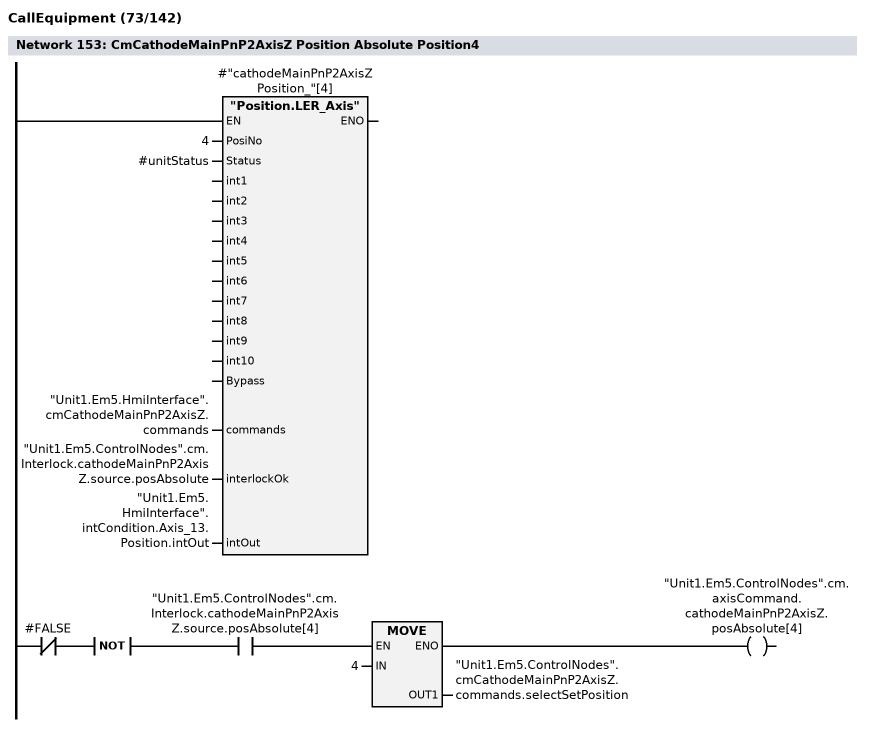
   RUNG wire#powerrail
      #"cathodeMainPnP2AxisZ Position_"[4](PosiNo := 4, Status := #unitStatus, int1 :=, int2 :=, int3 :=, int4 :=, int5 :=, int6 :=, int7 :=, int8 :=, int9 :=, int10 :=, Bypass :=, commands := "Unit1.Em5.HmiInterface".cmCathodeMainPnP2AxisZ.commands, interlockOk := "Unit1.Em5.ControlNodes".cm.Interlock.cathodeMainPnP2AxisZ.source.posAbsolute, intOut := "Unit1.Em5.HmiInterface".intCondition.Axis_13.Position.intOut)
   END_RUNG
   RUNG wire#powerrail
      I_Contact( #FALSE )
      Not()
      Contact( "Unit1.Em5.ControlNodes".cm.Interlock.cathodeMainPnP2AxisZ.source.posAbsolute[4] )
      Move(in := 4, out1 => "Unit1.Em5.ControlNodes".cmCathodeMainPnP2AxisZ.commands.selectSetPosition)
      Coil( "Unit1.Em5.ControlNodes".cm.axisCommand.cathodeMainPnP2AxisZ.posAbsolute[4] )
   END_RUNG
   // the same network as SCL:
   #"cathodeMainPnP2AxisZ Position_"[4](PosiNo := 4,   // "Position.LER_Axis"
                           Status := #unitStatus,
                           commands := "Unit1.Em5.HmiInterface".cmCathodeMainPnP2AxisZ.commands,
                           interlockOk := "Unit1.Em5.ControlNodes".cm.Interlock.cathodeMainPnP2AxisZ.source.posAbsolute,
                           intOut := "Unit1.Em5.HmiInterface".intCondition.Axis_13.Position.intOut);
   #_w1 := NOT (NOT #FALSE) AND "Unit1.Em5.ControlNodes".cm.Interlock.cathodeMainPnP2AxisZ.source.posAbsolute[4];
   IF #_w1 THEN "Unit1.Em5.ControlNodes".cmCathodeMainPnP2AxisZ.commands.selectSetPosition := 4; END_IF;
   "Unit1.Em5.ControlNodes".cm.axisCommand.cathodeMainPnP2AxisZ.posAbsolute[4] := #_w1;
END_REGION

REGION Network 154: CmCathodeMainPnP2AxisZ Position Absolute Position5
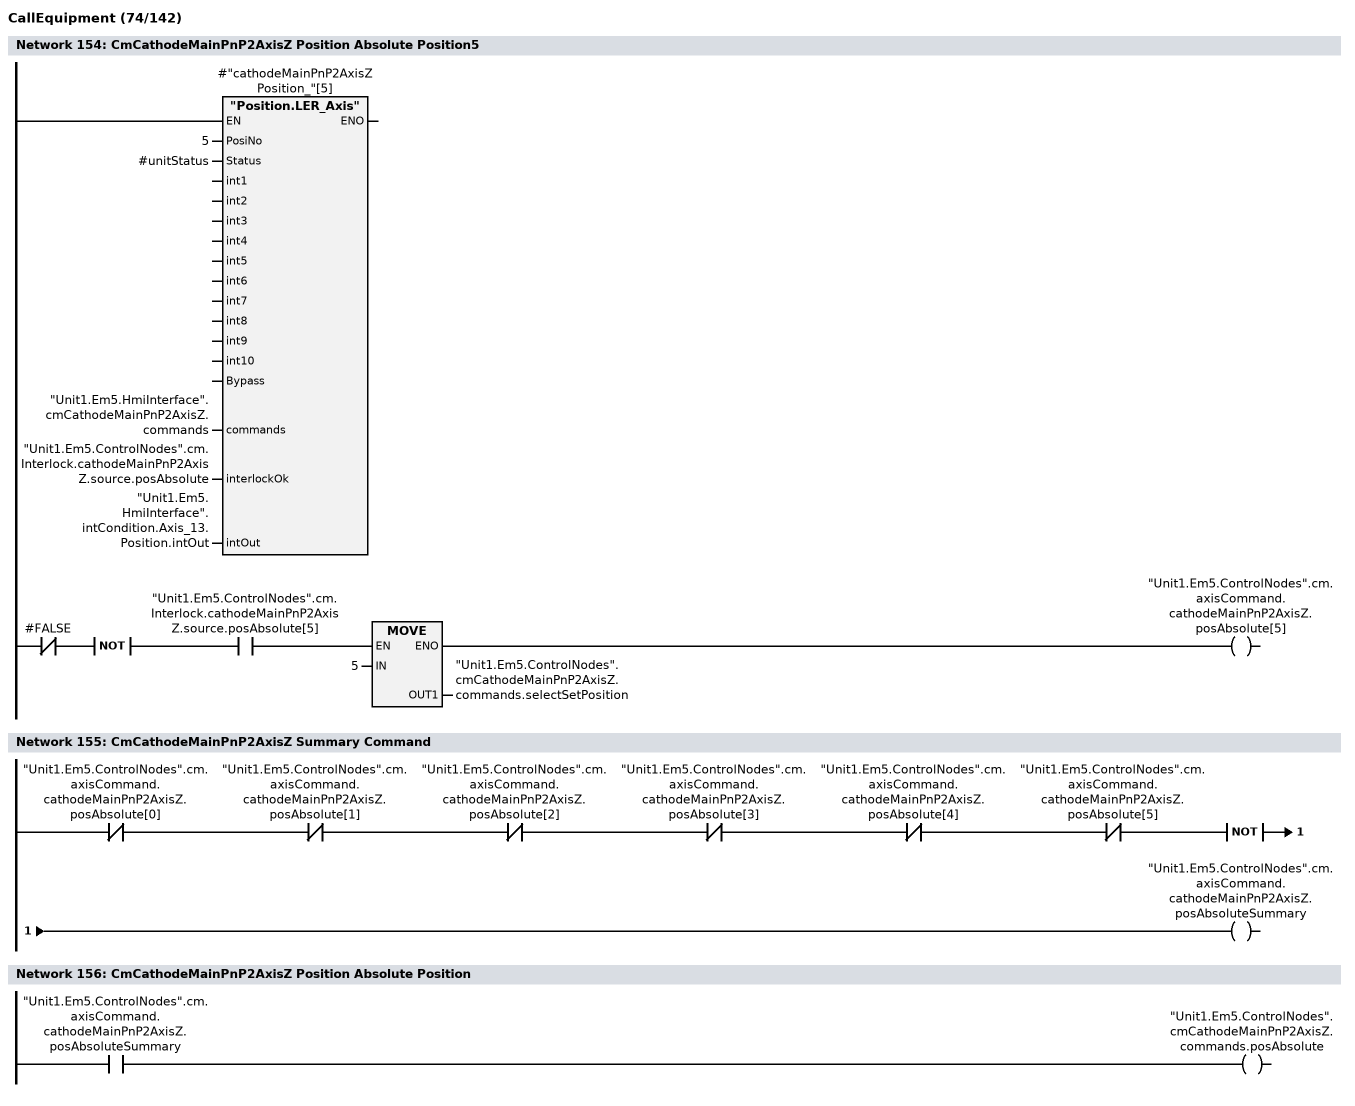
   RUNG wire#powerrail
      #"cathodeMainPnP2AxisZ Position_"[5](PosiNo := 5, Status := #unitStatus, int1 :=, int2 :=, int3 :=, int4 :=, int5 :=, int6 :=, int7 :=, int8 :=, int9 :=, int10 :=, Bypass :=, commands := "Unit1.Em5.HmiInterface".cmCathodeMainPnP2AxisZ.commands, interlockOk := "Unit1.Em5.ControlNodes".cm.Interlock.cathodeMainPnP2AxisZ.source.posAbsolute, intOut := "Unit1.Em5.HmiInterface".intCondition.Axis_13.Position.intOut)
   END_RUNG
   RUNG wire#powerrail
      I_Contact( #FALSE )
      Not()
      Contact( "Unit1.Em5.ControlNodes".cm.Interlock.cathodeMainPnP2AxisZ.source.posAbsolute[5] )
      Move(in := 5, out1 => "Unit1.Em5.ControlNodes".cmCathodeMainPnP2AxisZ.commands.selectSetPosition)
      Coil( "Unit1.Em5.ControlNodes".cm.axisCommand.cathodeMainPnP2AxisZ.posAbsolute[5] )
   END_RUNG
   // the same network as SCL:
   #"cathodeMainPnP2AxisZ Position_"[5](PosiNo := 5,   // "Position.LER_Axis"
                           Status := #unitStatus,
                           commands := "Unit1.Em5.HmiInterface".cmCathodeMainPnP2AxisZ.commands,
                           interlockOk := "Unit1.Em5.ControlNodes".cm.Interlock.cathodeMainPnP2AxisZ.source.posAbsolute,
                           intOut := "Unit1.Em5.HmiInterface".intCondition.Axis_13.Position.intOut);
   #_w1 := NOT (NOT #FALSE) AND "Unit1.Em5.ControlNodes".cm.Interlock.cathodeMainPnP2AxisZ.source.posAbsolute[5];
   IF #_w1 THEN "Unit1.Em5.ControlNodes".cmCathodeMainPnP2AxisZ.commands.selectSetPosition := 5; END_IF;
   "Unit1.Em5.ControlNodes".cm.axisCommand.cathodeMainPnP2AxisZ.posAbsolute[5] := #_w1;
END_REGION

REGION Network 155: CmCathodeMainPnP2AxisZ Summary Command
   RUNG wire#powerrail
      I_Contact( "Unit1.Em5.ControlNodes".cm.axisCommand.cathodeMainPnP2AxisZ.posAbsolute[0] )
      I_Contact( "Unit1.Em5.ControlNodes".cm.axisCommand.cathodeMainPnP2AxisZ.posAbsolute[1] )
      I_Contact( "Unit1.Em5.ControlNodes".cm.axisCommand.cathodeMainPnP2AxisZ.posAbsolute[2] )
      I_Contact( "Unit1.Em5.ControlNodes".cm.axisCommand.cathodeMainPnP2AxisZ.posAbsolute[3] )
      I_Contact( "Unit1.Em5.ControlNodes".cm.axisCommand.cathodeMainPnP2AxisZ.posAbsolute[4] )
      I_Contact( "Unit1.Em5.ControlNodes".cm.axisCommand.cathodeMainPnP2AxisZ.posAbsolute[5] )
      Not()
      Coil( "Unit1.Em5.ControlNodes".cm.axisCommand.cathodeMainPnP2AxisZ.posAbsoluteSummary )
   END_RUNG
   // the same network as SCL:
   "Unit1.Em5.ControlNodes".cm.axisCommand.cathodeMainPnP2AxisZ.posAbsoluteSummary := NOT (NOT "Unit1.Em5.ControlNodes".cm.axisCommand.cathodeMainPnP2AxisZ.posAbsolute[0] AND NOT "Unit1.Em5.ControlNodes".cm.axisCommand.cathodeMainPnP2AxisZ.posAbsolute[1] AND NOT "Unit1.Em5.ControlNodes".cm.axisCommand.cathodeMainPnP2AxisZ.posAbsolute[2] AND NOT "Unit1.Em5.ControlNodes".cm.axisCommand.cathodeMainPnP2AxisZ.posAbsolute[3] AND NOT "Unit1.Em5.ControlNodes".cm.axisCommand.cathodeMainPnP2AxisZ.posAbsolute[4] AND NOT "Unit1.Em5.ControlNodes".cm.axisCommand.cathodeMainPnP2AxisZ.posAbsolute[5]);
END_REGION

REGION Network 156: CmCathodeMainPnP2AxisZ Position Absolute Position
   RUNG wire#powerrail
      Contact( "Unit1.Em5.ControlNodes".cm.axisCommand.cathodeMainPnP2AxisZ.posAbsoluteSummary )
      Coil( "Unit1.Em5.ControlNodes".cmCathodeMainPnP2AxisZ.commands.posAbsolute )
   END_RUNG
   // the same network as SCL:
   "Unit1.Em5.ControlNodes".cmCathodeMainPnP2AxisZ.commands.posAbsolute := "Unit1.Em5.ControlNodes".cm.axisCommand.cathodeMainPnP2AxisZ.posAbsoluteSummary;
END_REGION

REGION Network 157: CmCathodeMainPnP1AxisZ Interlock Summary
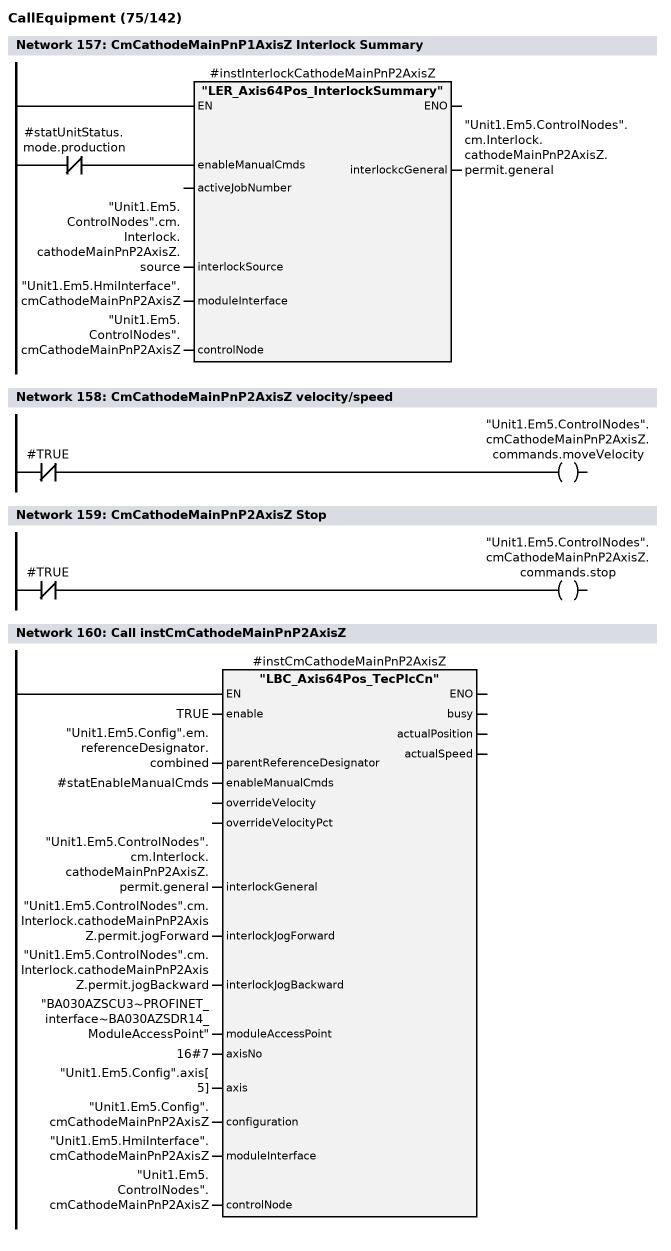
   RUNG wire#powerrail
      #instInterlockCathodeMainPnP2AxisZ(enableManualCmds := wire#w1, activeJobNumber :=, interlockSource := "Unit1.Em5.ControlNodes".cm.Interlock.cathodeMainPnP2AxisZ.source, moduleInterface := "Unit1.Em5.HmiInterface".cmCathodeMainPnP2AxisZ, controlNode := "Unit1.Em5.ControlNodes".cmCathodeMainPnP2AxisZ, interlockcGeneral => "Unit1.Em5.ControlNodes".cm.Interlock.cathodeMainPnP2AxisZ.permit.general)
   END_RUNG
   RUNG wire#powerrail
      I_Contact( #statUnitStatus.mode.production )
   END_RUNG wire#w1
   // the same network as SCL:
   #instInterlockCathodeMainPnP2AxisZ(enableManualCmds := NOT #statUnitStatus.mode.production,   // "LER_Axis64Pos_InterlockSummary"
                           interlockSource := "Unit1.Em5.ControlNodes".cm.Interlock.cathodeMainPnP2AxisZ.source,
                           moduleInterface := "Unit1.Em5.HmiInterface".cmCathodeMainPnP2AxisZ,
                           controlNode := "Unit1.Em5.ControlNodes".cmCathodeMainPnP2AxisZ,
                           interlockcGeneral => "Unit1.Em5.ControlNodes".cm.Interlock.cathodeMainPnP2AxisZ.permit.general);
END_REGION

REGION Network 158: CmCathodeMainPnP2AxisZ velocity/speed
   RUNG wire#powerrail
      I_Contact( #TRUE )
      Coil( "Unit1.Em5.ControlNodes".cmCathodeMainPnP2AxisZ.commands.moveVelocity )
   END_RUNG
   // the same network as SCL:
   "Unit1.Em5.ControlNodes".cmCathodeMainPnP2AxisZ.commands.moveVelocity := NOT #TRUE;
END_REGION

REGION Network 159: CmCathodeMainPnP2AxisZ Stop
   RUNG wire#powerrail
      I_Contact( #TRUE )
      Coil( "Unit1.Em5.ControlNodes".cmCathodeMainPnP2AxisZ.commands.stop )
   END_RUNG
   // the same network as SCL:
   "Unit1.Em5.ControlNodes".cmCathodeMainPnP2AxisZ.commands.stop := NOT #TRUE;
END_REGION

REGION Network 160: Call instCmCathodeMainPnP2AxisZ
   RUNG wire#powerrail
      #instCmCathodeMainPnP2AxisZ(enable := TRUE, parentReferenceDesignator := "Unit1.Em5.Config".em.referenceDesignator.combined, enableManualCmds := #statEnableManualCmds, overrideVelocity :=, overrideVelocityPct :=, interlockGeneral := "Unit1.Em5.ControlNodes".cm.Interlock.cathodeMainPnP2AxisZ.permit.general, interlockJogForward := "Unit1.Em5.ControlNodes".cm.Interlock.cathodeMainPnP2AxisZ.permit.jogForward, interlockJogBackward := "Unit1.Em5.ControlNodes".cm.Interlock.cathodeMainPnP2AxisZ.permit.jogBackward, moduleAccessPoint := "BA030AZSCU3~PROFINET_interface~BA030AZSDR14_ModuleAccessPoint", axisNo := 16#7, axis := "Unit1.Em5.Config".axis[5], configuration := "Unit1.Em5.Config".cmCathodeMainPnP2AxisZ, moduleInterface := "Unit1.Em5.HmiInterface".cmCathodeMainPnP2AxisZ, controlNode := "Unit1.Em5.ControlNodes".cmCathodeMainPnP2AxisZ, busy =>, actualPosition =>, actualSpeed =>)
   END_RUNG
   // the same network as SCL:
   #instCmCathodeMainPnP2AxisZ(enable := TRUE,   // "LBC_Axis64Pos_TecPlcCn"
                           parentReferenceDesignator := "Unit1.Em5.Config".em.referenceDesignator.combined,
                           enableManualCmds := #statEnableManualCmds,
                           interlockGeneral := "Unit1.Em5.ControlNodes".cm.Interlock.cathodeMainPnP2AxisZ.permit.general,
                           interlockJogForward := "Unit1.Em5.ControlNodes".cm.Interlock.cathodeMainPnP2AxisZ.permit.jogForward,
                           interlockJogBackward := "Unit1.Em5.ControlNodes".cm.Interlock.cathodeMainPnP2AxisZ.permit.jogBackward,
                           moduleAccessPoint := "BA030AZSCU3~PROFINET_interface~BA030AZSDR14_ModuleAccessPoint",
                           axisNo := 16#7,
                           axis := "Unit1.Em5.Config".axis[5],
                           configuration := "Unit1.Em5.Config".cmCathodeMainPnP2AxisZ,
                           moduleInterface := "Unit1.Em5.HmiInterface".cmCathodeMainPnP2AxisZ,
                           controlNode := "Unit1.Em5.ControlNodes".cmCathodeMainPnP2AxisZ);
END_REGION

REGION Network 161: CmCathodeMainPnP2AxisY SoftCam
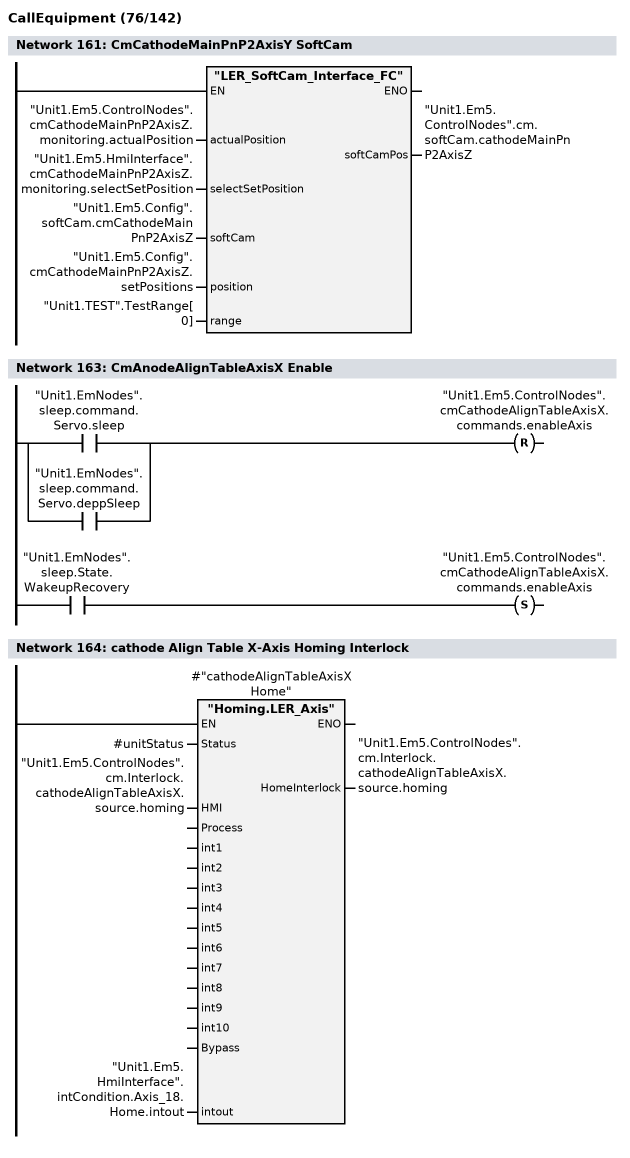
   RUNG wire#powerrail
      "LER_SoftCam_Interface_FC"(actualPosition := "Unit1.Em5.ControlNodes".cmCathodeMainPnP2AxisZ.monitoring.actualPosition, selectSetPosition := "Unit1.Em5.HmiInterface".cmCathodeMainPnP2AxisZ.monitoring.selectSetPosition, softCam := "Unit1.Em5.Config".softCam.cmCathodeMainPnP2AxisZ, position := "Unit1.Em5.Config".cmCathodeMainPnP2AxisZ.setPositions, range := "Unit1.TEST".TestRange[0], softCamPos => "Unit1.Em5.ControlNodes".cm.softCam.cathodeMainPnP2AxisZ)
   END_RUNG
   // the same network as SCL:
   "LER_SoftCam_Interface_FC"(actualPosition := "Unit1.Em5.ControlNodes".cmCathodeMainPnP2AxisZ.monitoring.actualPosition,
                           selectSetPosition := "Unit1.Em5.HmiInterface".cmCathodeMainPnP2AxisZ.monitoring.selectSetPosition,
                           softCam := "Unit1.Em5.Config".softCam.cmCathodeMainPnP2AxisZ,
                           position := "Unit1.Em5.Config".cmCathodeMainPnP2AxisZ.setPositions,
                           range := "Unit1.TEST".TestRange[0],
                           softCamPos => "Unit1.Em5.ControlNodes".cm.softCam.cathodeMainPnP2AxisZ);
END_REGION

REGION Network 163: CmAnodeAlignTableAxisX Enable
   RUNG wire#powerrail
      Contact( "Unit1.EmNodes".sleep.command.Servo.sleep )
      wire#w1
      R_Coil( "Unit1.Em5.ControlNodes".cmCathodeAlignTableAxisX.commands.enableAxis )
   END_RUNG
   RUNG wire#powerrail
      Contact( "Unit1.EmNodes".sleep.command.Servo.deppSleep )
   END_RUNG wire#w1
   RUNG wire#powerrail
      Contact( "Unit1.EmNodes".sleep.State.WakeupRecovery )
      S_Coil( "Unit1.Em5.ControlNodes".cmCathodeAlignTableAxisX.commands.enableAxis )
   END_RUNG
   // the same network as SCL:
   IF "Unit1.EmNodes".sleep.command.Servo.sleep OR "Unit1.EmNodes".sleep.command.Servo.deppSleep THEN
       "Unit1.Em5.ControlNodes".cmCathodeAlignTableAxisX.commands.enableAxis := FALSE;
   END_IF;
   IF "Unit1.EmNodes".sleep.State.WakeupRecovery THEN
       "Unit1.Em5.ControlNodes".cmCathodeAlignTableAxisX.commands.enableAxis := TRUE;
   END_IF;
END_REGION

REGION Network 164: cathode Align Table X-Axis Homing Interlock
   RUNG wire#powerrail
      #"cathodeAlignTableAxisX Home"(Status := #unitStatus, HMI := "Unit1.Em5.ControlNodes".cm.Interlock.cathodeAlignTableAxisX.source.homing, Process :=, int1 :=, int2 :=, int3 :=, int4 :=, int5 :=, int6 :=, int7 :=, int8 :=, int9 :=, int10 :=, Bypass :=, intout := "Unit1.Em5.HmiInterface".intCondition.Axis_18.Home.intout, HomeInterlock => "Unit1.Em5.ControlNodes".cm.Interlock.cathodeAlignTableAxisX.source.homing)
   END_RUNG
   // the same network as SCL:
   #"cathodeAlignTableAxisX Home"(Status := #unitStatus,   // "Homing.LER_Axis"
                           HMI := "Unit1.Em5.ControlNodes".cm.Interlock.cathodeAlignTableAxisX.source.homing,
                           intout := "Unit1.Em5.HmiInterface".intCondition.Axis_18.Home.intout,
                           HomeInterlock => "Unit1.Em5.ControlNodes".cm.Interlock.cathodeAlignTableAxisX.source.homing);
END_REGION

REGION Network 165: CmCathodeAlignTableAxisX Position Absolute Jog
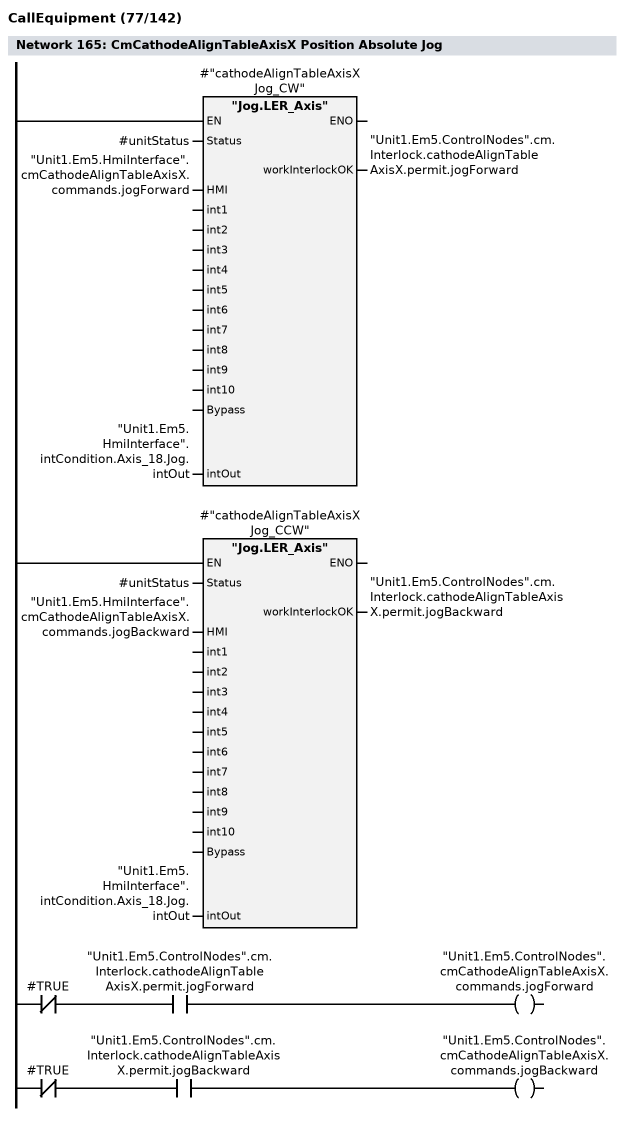
   RUNG wire#powerrail
      #"cathodeAlignTableAxisX Jog_CW"(Status := #unitStatus, HMI := "Unit1.Em5.HmiInterface".cmCathodeAlignTableAxisX.commands.jogForward, int1 :=, int2 :=, int3 :=, int4 :=, int5 :=, int6 :=, int7 :=, int8 :=, int9 :=, int10 :=, Bypass :=, intOut := "Unit1.Em5.HmiInterface".intCondition.Axis_18.Jog.intOut, workInterlockOK => "Unit1.Em5.ControlNodes".cm.Interlock.cathodeAlignTableAxisX.permit.jogForward)
   END_RUNG
   RUNG wire#powerrail
      #"cathodeAlignTableAxisX Jog_CCW"(Status := #unitStatus, HMI := "Unit1.Em5.HmiInterface".cmCathodeAlignTableAxisX.commands.jogBackward, int1 :=, int2 :=, int3 :=, int4 :=, int5 :=, int6 :=, int7 :=, int8 :=, int9 :=, int10 :=, Bypass :=, intOut := "Unit1.Em5.HmiInterface".intCondition.Axis_18.Jog.intOut, workInterlockOK => "Unit1.Em5.ControlNodes".cm.Interlock.cathodeAlignTableAxisX.permit.jogBackward)
   END_RUNG
   RUNG wire#powerrail
      I_Contact( #TRUE )
      Contact( "Unit1.Em5.ControlNodes".cm.Interlock.cathodeAlignTableAxisX.permit.jogForward )
      Coil( "Unit1.Em5.ControlNodes".cmCathodeAlignTableAxisX.commands.jogForward )
   END_RUNG
   RUNG wire#powerrail
      I_Contact( #TRUE )
      Contact( "Unit1.Em5.ControlNodes".cm.Interlock.cathodeAlignTableAxisX.permit.jogBackward )
      Coil( "Unit1.Em5.ControlNodes".cmCathodeAlignTableAxisX.commands.jogBackward )
   END_RUNG
   // the same network as SCL:
   #"cathodeAlignTableAxisX Jog_CW"(Status := #unitStatus,   // "Jog.LER_Axis"
                           HMI := "Unit1.Em5.HmiInterface".cmCathodeAlignTableAxisX.commands.jogForward,
                           intOut := "Unit1.Em5.HmiInterface".intCondition.Axis_18.Jog.intOut,
                           workInterlockOK => "Unit1.Em5.ControlNodes".cm.Interlock.cathodeAlignTableAxisX.permit.jogForward);
   #"cathodeAlignTableAxisX Jog_CCW"(Status := #unitStatus,   // "Jog.LER_Axis"
                           HMI := "Unit1.Em5.HmiInterface".cmCathodeAlignTableAxisX.commands.jogBackward,
                           intOut := "Unit1.Em5.HmiInterface".intCondition.Axis_18.Jog.intOut,
                           workInterlockOK => "Unit1.Em5.ControlNodes".cm.Interlock.cathodeAlignTableAxisX.permit.jogBackward);
   "Unit1.Em5.ControlNodes".cmCathodeAlignTableAxisX.commands.jogForward := NOT #TRUE AND "Unit1.Em5.ControlNodes".cm.Interlock.cathodeAlignTableAxisX.permit.jogForward;
   "Unit1.Em5.ControlNodes".cmCathodeAlignTableAxisX.commands.jogBackward := NOT #TRUE AND "Unit1.Em5.ControlNodes".cm.Interlock.cathodeAlignTableAxisX.permit.jogBackward;
END_REGION

REGION Network 166: CmCathodeAlignTableAxisX Position Absolute Position0
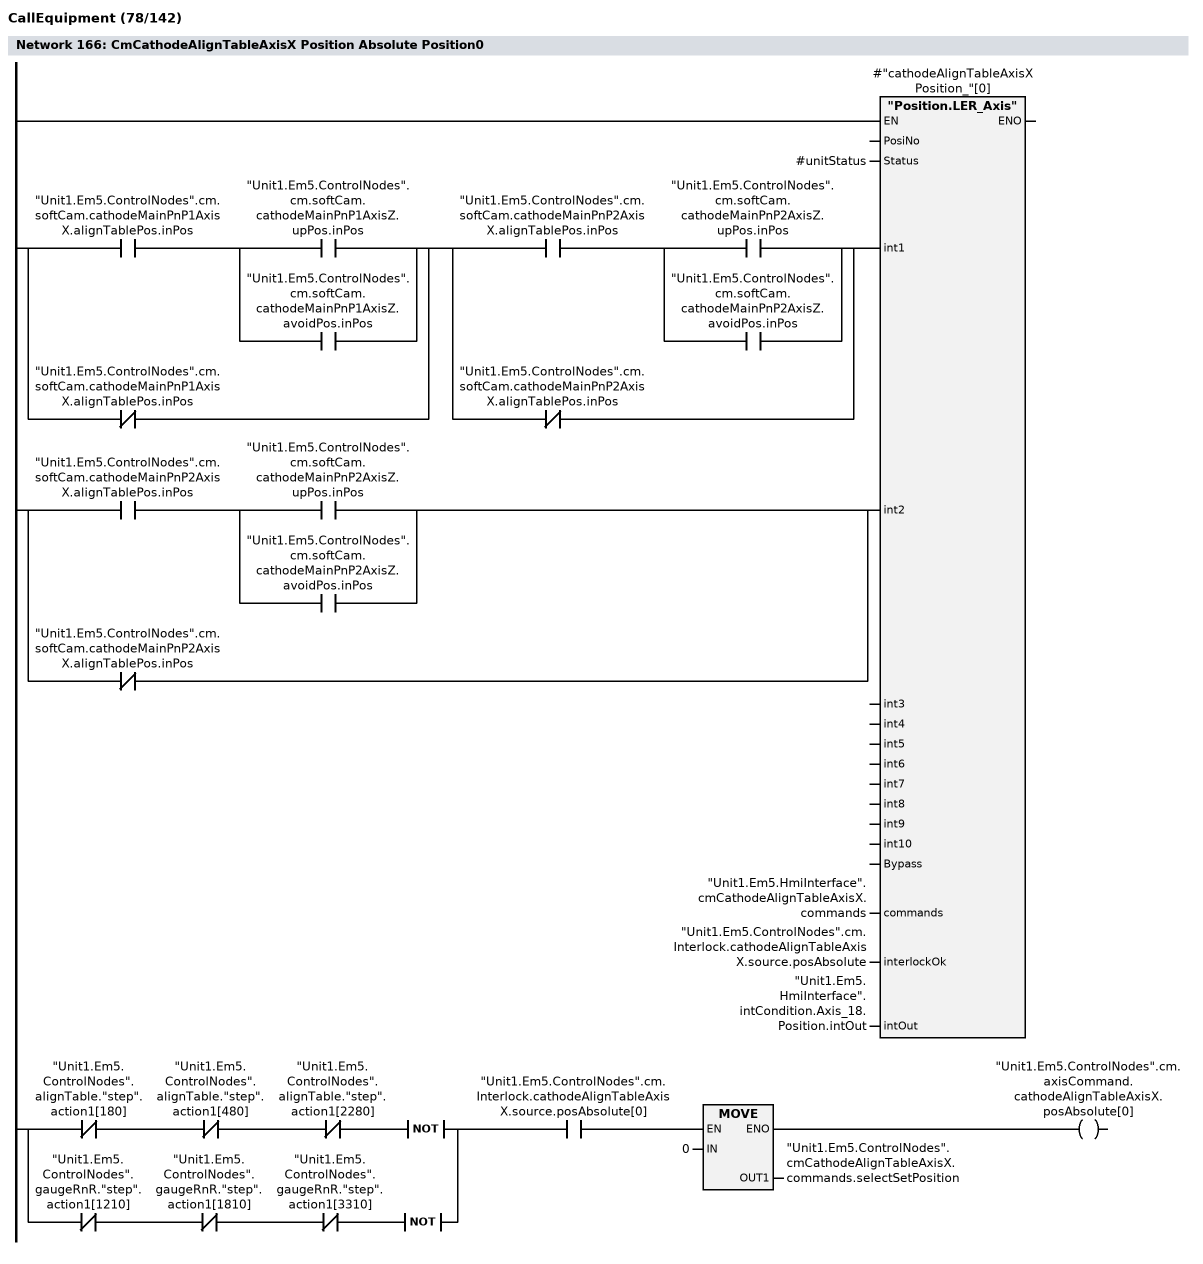
   RUNG wire#powerrail
      #"cathodeAlignTableAxisX Position_"[0](int1 := wire#w4, int2 := wire#w6, PosiNo :=, Status := #unitStatus, int3 :=, int4 :=, int5 :=, int6 :=, int7 :=, int8 :=, int9 :=, int10 :=, Bypass :=, commands := "Unit1.Em5.HmiInterface".cmCathodeAlignTableAxisX.commands, interlockOk := "Unit1.Em5.ControlNodes".cm.Interlock.cathodeAlignTableAxisX.source.posAbsolute, intOut := "Unit1.Em5.HmiInterface".intCondition.Axis_18.Position.intOut)
   END_RUNG
   RUNG wire#powerrail
      Contact( "Unit1.Em5.ControlNodes".cm.softCam.cathodeMainPnP1AxisX.alignTablePos.inPos )
      wire#w1
      Contact( "Unit1.Em5.ControlNodes".cm.softCam.cathodeMainPnP1AxisZ.upPos.inPos )
      wire#w2
      Contact( "Unit1.Em5.ControlNodes".cm.softCam.cathodeMainPnP2AxisX.alignTablePos.inPos )
      wire#w3
      Contact( "Unit1.Em5.ControlNodes".cm.softCam.cathodeMainPnP2AxisZ.upPos.inPos )
   END_RUNG wire#w4
   RUNG wire#w1
      Contact( "Unit1.Em5.ControlNodes".cm.softCam.cathodeMainPnP1AxisZ.avoidPos.inPos )
   END_RUNG wire#w2
   RUNG wire#powerrail
      I_Contact( "Unit1.Em5.ControlNodes".cm.softCam.cathodeMainPnP1AxisX.alignTablePos.inPos )
   END_RUNG wire#w2
   RUNG wire#w3
      Contact( "Unit1.Em5.ControlNodes".cm.softCam.cathodeMainPnP2AxisZ.avoidPos.inPos )
   END_RUNG wire#w4
   RUNG wire#w2
      I_Contact( "Unit1.Em5.ControlNodes".cm.softCam.cathodeMainPnP2AxisX.alignTablePos.inPos )
   END_RUNG wire#w4
   RUNG wire#powerrail
      Contact( "Unit1.Em5.ControlNodes".cm.softCam.cathodeMainPnP2AxisX.alignTablePos.inPos )
      wire#w5
      Contact( "Unit1.Em5.ControlNodes".cm.softCam.cathodeMainPnP2AxisZ.upPos.inPos )
   END_RUNG wire#w6
   RUNG wire#w5
      Contact( "Unit1.Em5.ControlNodes".cm.softCam.cathodeMainPnP2AxisZ.avoidPos.inPos )
   END_RUNG wire#w6
   RUNG wire#powerrail
      I_Contact( "Unit1.Em5.ControlNodes".cm.softCam.cathodeMainPnP2AxisX.alignTablePos.inPos )
   END_RUNG wire#w6
   RUNG wire#powerrail
      I_Contact( "Unit1.Em5.ControlNodes".alignTable."step".action1[180] )
      I_Contact( "Unit1.Em5.ControlNodes".alignTable."step".action1[480] )
      I_Contact( "Unit1.Em5.ControlNodes".alignTable."step".action1[2280] )
      Not()
      wire#w7
      Contact( "Unit1.Em5.ControlNodes".cm.Interlock.cathodeAlignTableAxisX.source.posAbsolute[0] )
      Move(in := 0, out1 => "Unit1.Em5.ControlNodes".cmCathodeAlignTableAxisX.commands.selectSetPosition)
      Coil( "Unit1.Em5.ControlNodes".cm.axisCommand.cathodeAlignTableAxisX.posAbsolute[0] )
   END_RUNG
   RUNG wire#powerrail
      I_Contact( "Unit1.Em5.ControlNodes".gaugeRnR."step".action1[1210] )
      I_Contact( "Unit1.Em5.ControlNodes".gaugeRnR."step".action1[1810] )
      I_Contact( "Unit1.Em5.ControlNodes".gaugeRnR."step".action1[3310] )
      Not()
   END_RUNG wire#w7
   // the same network as SCL:
   #"cathodeAlignTableAxisX Position_"[0](Status := #unitStatus,   // "Position.LER_Axis"
                           int1 := (("Unit1.Em5.ControlNodes".cm.softCam.cathodeMainPnP1AxisX.alignTablePos.inPos AND ("Unit1.Em5.ControlNodes".cm.softCam.cathodeMainPnP1AxisZ.upPos.inPos OR "Unit1.Em5.ControlNodes".cm.softCam.cathodeMainPnP1AxisZ.avoidPos.inPos)) OR NOT "Unit1.Em5.ControlNodes".cm.softCam.cathodeMainPnP1AxisX.alignTablePos.inPos) AND (("Unit1.Em5.ControlNodes".cm.softCam.cathodeMainPnP2AxisX.alignTablePos.inPos AND ("Unit1.Em5.ControlNodes".cm.softCam.cathodeMainPnP2AxisZ.upPos.inPos OR "Unit1.Em5.ControlNodes".cm.softCam.cathodeMainPnP2AxisZ.avoidPos.inPos)) OR NOT "Unit1.Em5.ControlNodes".cm.softCam.cathodeMainPnP2AxisX.alignTablePos.inPos),
                           int2 := ("Unit1.Em5.ControlNodes".cm.softCam.cathodeMainPnP2AxisX.alignTablePos.inPos AND ("Unit1.Em5.ControlNodes".cm.softCam.cathodeMainPnP2AxisZ.upPos.inPos OR "Unit1.Em5.ControlNodes".cm.softCam.cathodeMainPnP2AxisZ.avoidPos.inPos)) OR NOT "Unit1.Em5.ControlNodes".cm.softCam.cathodeMainPnP2AxisX.alignTablePos.inPos,
                           commands := "Unit1.Em5.HmiInterface".cmCathodeAlignTableAxisX.commands,
                           interlockOk := "Unit1.Em5.ControlNodes".cm.Interlock.cathodeAlignTableAxisX.source.posAbsolute,
                           intOut := "Unit1.Em5.HmiInterface".intCondition.Axis_18.Position.intOut);
   #_w1 := (NOT (NOT "Unit1.Em5.ControlNodes".alignTable."step".action1[180] AND NOT "Unit1.Em5.ControlNodes".alignTable."step".action1[480] AND NOT "Unit1.Em5.ControlNodes".alignTable."step".action1[2280]) OR NOT (NOT "Unit1.Em5.ControlNodes".gaugeRnR."step".action1[1210] AND NOT "Unit1.Em5.ControlNodes".gaugeRnR."step".action1[1810] AND NOT "Unit1.Em5.ControlNodes".gaugeRnR."step".action1[3310])) AND "Unit1.Em5.ControlNodes".cm.Interlock.cathodeAlignTableAxisX.source.posAbsolute[0];
   IF #_w1 THEN "Unit1.Em5.ControlNodes".cmCathodeAlignTableAxisX.commands.selectSetPosition := 0; END_IF;
   "Unit1.Em5.ControlNodes".cm.axisCommand.cathodeAlignTableAxisX.posAbsolute[0] := #_w1;
END_REGION

REGION Network 167: CmCathodeAlignTableAxisX Position Absolute Position1
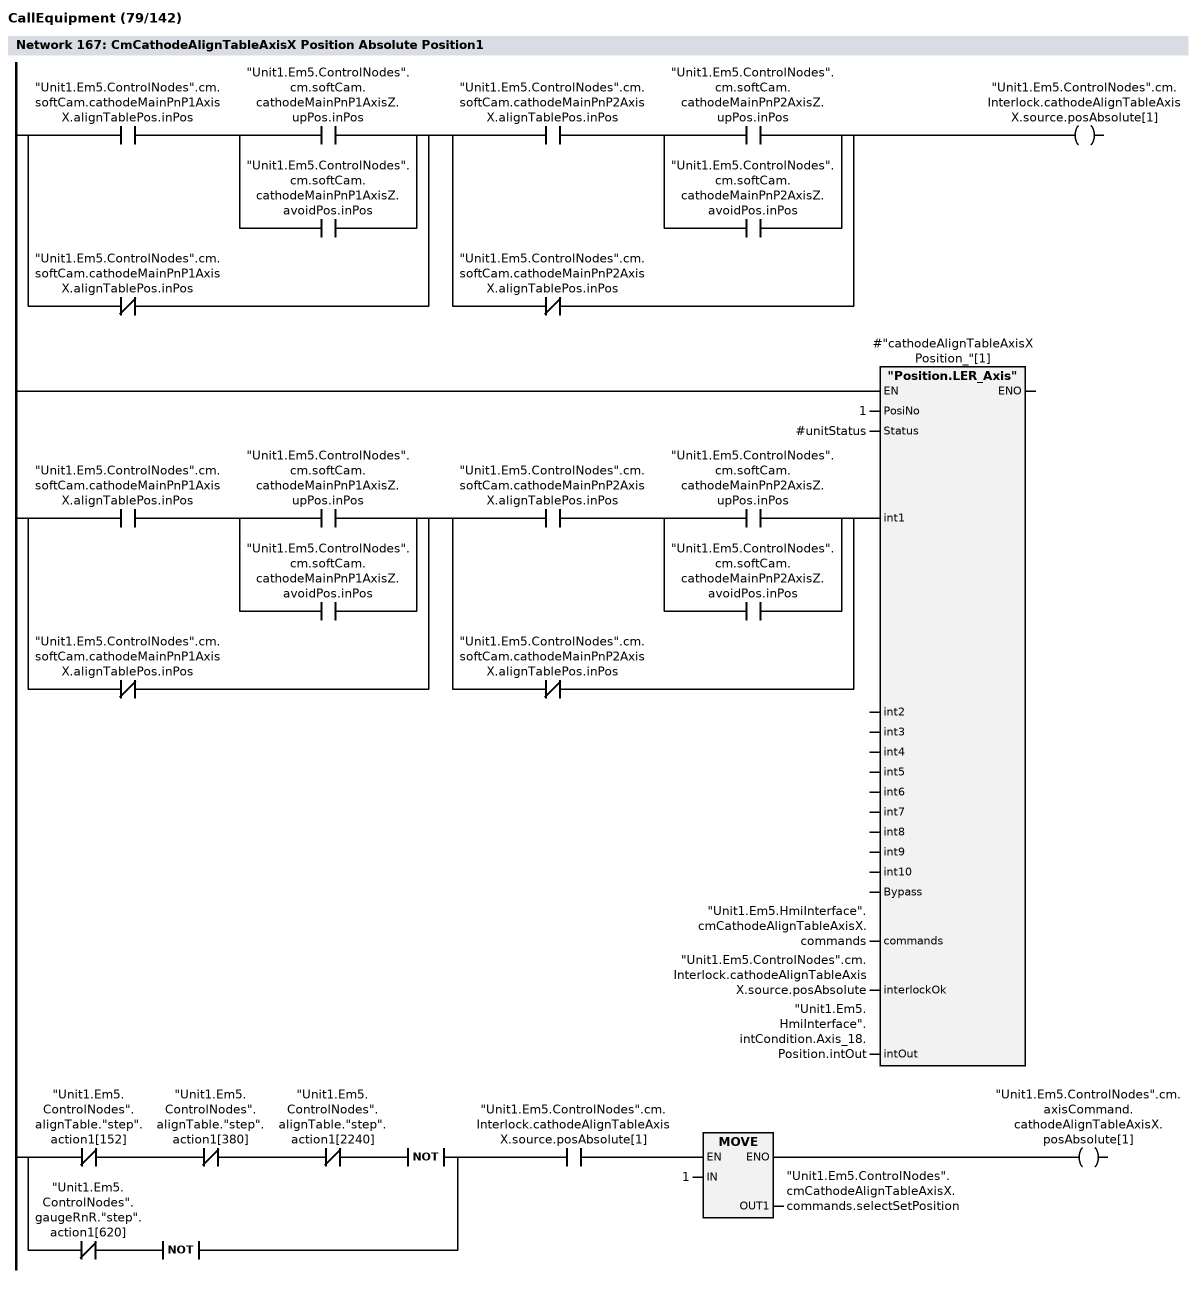
   RUNG wire#powerrail
      Contact( "Unit1.Em5.ControlNodes".cm.softCam.cathodeMainPnP1AxisX.alignTablePos.inPos )
      wire#w1
      Contact( "Unit1.Em5.ControlNodes".cm.softCam.cathodeMainPnP1AxisZ.upPos.inPos )
      wire#w2
      Contact( "Unit1.Em5.ControlNodes".cm.softCam.cathodeMainPnP2AxisX.alignTablePos.inPos )
      wire#w3
      Contact( "Unit1.Em5.ControlNodes".cm.softCam.cathodeMainPnP2AxisZ.upPos.inPos )
      wire#w4
      Coil( "Unit1.Em5.ControlNodes".cm.Interlock.cathodeAlignTableAxisX.source.posAbsolute[1] )
   END_RUNG
   RUNG wire#w1
      Contact( "Unit1.Em5.ControlNodes".cm.softCam.cathodeMainPnP1AxisZ.avoidPos.inPos )
   END_RUNG wire#w2
   RUNG wire#powerrail
      I_Contact( "Unit1.Em5.ControlNodes".cm.softCam.cathodeMainPnP1AxisX.alignTablePos.inPos )
   END_RUNG wire#w2
   RUNG wire#w3
      Contact( "Unit1.Em5.ControlNodes".cm.softCam.cathodeMainPnP2AxisZ.avoidPos.inPos )
   END_RUNG wire#w4
   RUNG wire#w2
      I_Contact( "Unit1.Em5.ControlNodes".cm.softCam.cathodeMainPnP2AxisX.alignTablePos.inPos )
   END_RUNG wire#w4
   RUNG wire#powerrail
      #"cathodeAlignTableAxisX Position_"[1](int1 := wire#w8, PosiNo := 1, Status := #unitStatus, int2 :=, int3 :=, int4 :=, int5 :=, int6 :=, int7 :=, int8 :=, int9 :=, int10 :=, Bypass :=, commands := "Unit1.Em5.HmiInterface".cmCathodeAlignTableAxisX.commands, interlockOk := "Unit1.Em5.ControlNodes".cm.Interlock.cathodeAlignTableAxisX.source.posAbsolute, intOut := "Unit1.Em5.HmiInterface".intCondition.Axis_18.Position.intOut)
   END_RUNG
   RUNG wire#powerrail
      Contact( "Unit1.Em5.ControlNodes".cm.softCam.cathodeMainPnP1AxisX.alignTablePos.inPos )
      wire#w5
      Contact( "Unit1.Em5.ControlNodes".cm.softCam.cathodeMainPnP1AxisZ.upPos.inPos )
      wire#w6
      Contact( "Unit1.Em5.ControlNodes".cm.softCam.cathodeMainPnP2AxisX.alignTablePos.inPos )
      wire#w7
      Contact( "Unit1.Em5.ControlNodes".cm.softCam.cathodeMainPnP2AxisZ.upPos.inPos )
   END_RUNG wire#w8
   RUNG wire#w5
      Contact( "Unit1.Em5.ControlNodes".cm.softCam.cathodeMainPnP1AxisZ.avoidPos.inPos )
   END_RUNG wire#w6
   RUNG wire#powerrail
      I_Contact( "Unit1.Em5.ControlNodes".cm.softCam.cathodeMainPnP1AxisX.alignTablePos.inPos )
   END_RUNG wire#w6
   RUNG wire#w7
      Contact( "Unit1.Em5.ControlNodes".cm.softCam.cathodeMainPnP2AxisZ.avoidPos.inPos )
   END_RUNG wire#w8
   RUNG wire#w6
      I_Contact( "Unit1.Em5.ControlNodes".cm.softCam.cathodeMainPnP2AxisX.alignTablePos.inPos )
   END_RUNG wire#w8
   RUNG wire#powerrail
      I_Contact( "Unit1.Em5.ControlNodes".alignTable."step".action1[152] )
      I_Contact( "Unit1.Em5.ControlNodes".alignTable."step".action1[380] )
      I_Contact( "Unit1.Em5.ControlNodes".alignTable."step".action1[2240] )
      Not()
      wire#w9
      Contact( "Unit1.Em5.ControlNodes".cm.Interlock.cathodeAlignTableAxisX.source.posAbsolute[1] )
      Move(in := 1, out1 => "Unit1.Em5.ControlNodes".cmCathodeAlignTableAxisX.commands.selectSetPosition)
      Coil( "Unit1.Em5.ControlNodes".cm.axisCommand.cathodeAlignTableAxisX.posAbsolute[1] )
   END_RUNG
   RUNG wire#powerrail
      I_Contact( "Unit1.Em5.ControlNodes".gaugeRnR."step".action1[620] )
      Not()
   END_RUNG wire#w9
   // the same network as SCL:
   "Unit1.Em5.ControlNodes".cm.Interlock.cathodeAlignTableAxisX.source.posAbsolute[1] := (("Unit1.Em5.ControlNodes".cm.softCam.cathodeMainPnP1AxisX.alignTablePos.inPos AND ("Unit1.Em5.ControlNodes".cm.softCam.cathodeMainPnP1AxisZ.upPos.inPos OR "Unit1.Em5.ControlNodes".cm.softCam.cathodeMainPnP1AxisZ.avoidPos.inPos)) OR NOT "Unit1.Em5.ControlNodes".cm.softCam.cathodeMainPnP1AxisX.alignTablePos.inPos) AND (("Unit1.Em5.ControlNodes".cm.softCam.cathodeMainPnP2AxisX.alignTablePos.inPos AND ("Unit1.Em5.ControlNodes".cm.softCam.cathodeMainPnP2AxisZ.upPos.inPos OR "Unit1.Em5.ControlNodes".cm.softCam.cathodeMainPnP2AxisZ.avoidPos.inPos)) OR NOT "Unit1.Em5.ControlNodes".cm.softCam.cathodeMainPnP2AxisX.alignTablePos.inPos);
   #"cathodeAlignTableAxisX Position_"[1](PosiNo := 1,   // "Position.LER_Axis"
                           Status := #unitStatus,
                           int1 := (("Unit1.Em5.ControlNodes".cm.softCam.cathodeMainPnP1AxisX.alignTablePos.inPos AND ("Unit1.Em5.ControlNodes".cm.softCam.cathodeMainPnP1AxisZ.upPos.inPos OR "Unit1.Em5.ControlNodes".cm.softCam.cathodeMainPnP1AxisZ.avoidPos.inPos)) OR NOT "Unit1.Em5.ControlNodes".cm.softCam.cathodeMainPnP1AxisX.alignTablePos.inPos) AND (("Unit1.Em5.ControlNodes".cm.softCam.cathodeMainPnP2AxisX.alignTablePos.inPos AND ("Unit1.Em5.ControlNodes".cm.softCam.cathodeMainPnP2AxisZ.upPos.inPos OR "Unit1.Em5.ControlNodes".cm.softCam.cathodeMainPnP2AxisZ.avoidPos.inPos)) OR NOT "Unit1.Em5.ControlNodes".cm.softCam.cathodeMainPnP2AxisX.alignTablePos.inPos),
                           commands := "Unit1.Em5.HmiInterface".cmCathodeAlignTableAxisX.commands,
                           interlockOk := "Unit1.Em5.ControlNodes".cm.Interlock.cathodeAlignTableAxisX.source.posAbsolute,
                           intOut := "Unit1.Em5.HmiInterface".intCondition.Axis_18.Position.intOut);
   #_w1 := (NOT (NOT "Unit1.Em5.ControlNodes".alignTable."step".action1[152] AND NOT "Unit1.Em5.ControlNodes".alignTable."step".action1[380] AND NOT "Unit1.Em5.ControlNodes".alignTable."step".action1[2240]) OR NOT (NOT "Unit1.Em5.ControlNodes".gaugeRnR."step".action1[620])) AND "Unit1.Em5.ControlNodes".cm.Interlock.cathodeAlignTableAxisX.source.posAbsolute[1];
   IF #_w1 THEN "Unit1.Em5.ControlNodes".cmCathodeAlignTableAxisX.commands.selectSetPosition := 1; END_IF;
   "Unit1.Em5.ControlNodes".cm.axisCommand.cathodeAlignTableAxisX.posAbsolute[1] := #_w1;
END_REGION

REGION Network 168: CmCathodeAlignTableAxisX Position Absolute Position2
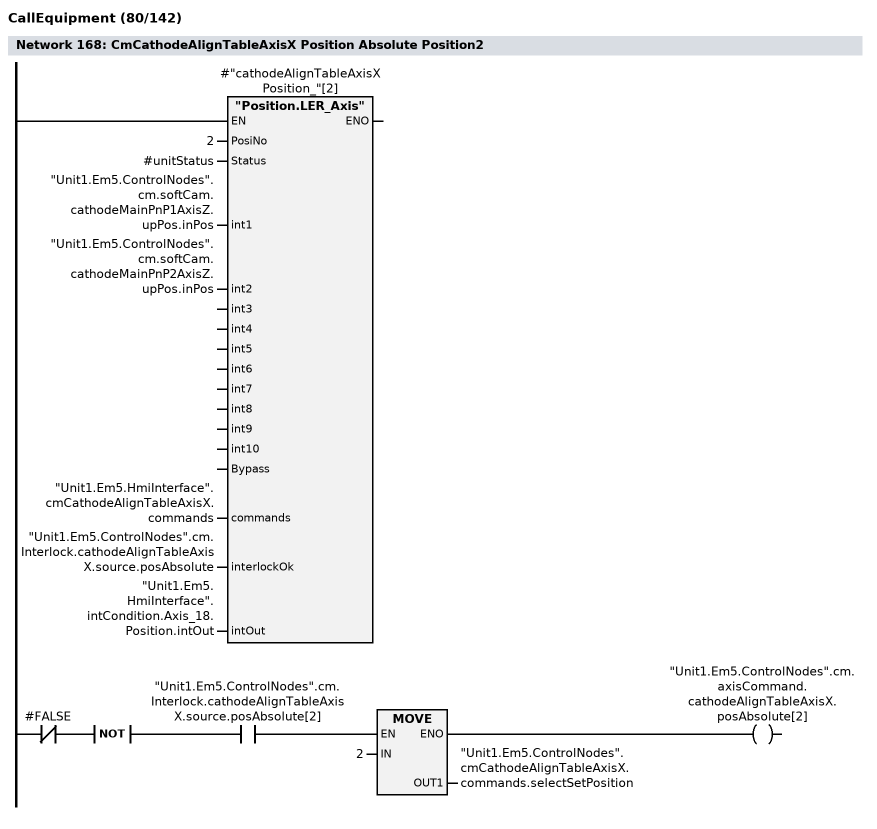
   RUNG wire#powerrail
      #"cathodeAlignTableAxisX Position_"[2](PosiNo := 2, Status := #unitStatus, int1 := "Unit1.Em5.ControlNodes".cm.softCam.cathodeMainPnP1AxisZ.upPos.inPos, int2 := "Unit1.Em5.ControlNodes".cm.softCam.cathodeMainPnP2AxisZ.upPos.inPos, int3 :=, int4 :=, int5 :=, int6 :=, int7 :=, int8 :=, int9 :=, int10 :=, Bypass :=, commands := "Unit1.Em5.HmiInterface".cmCathodeAlignTableAxisX.commands, interlockOk := "Unit1.Em5.ControlNodes".cm.Interlock.cathodeAlignTableAxisX.source.posAbsolute, intOut := "Unit1.Em5.HmiInterface".intCondition.Axis_18.Position.intOut)
   END_RUNG
   RUNG wire#powerrail
      I_Contact( #FALSE )
      Not()
      Contact( "Unit1.Em5.ControlNodes".cm.Interlock.cathodeAlignTableAxisX.source.posAbsolute[2] )
      Move(in := 2, out1 => "Unit1.Em5.ControlNodes".cmCathodeAlignTableAxisX.commands.selectSetPosition)
      Coil( "Unit1.Em5.ControlNodes".cm.axisCommand.cathodeAlignTableAxisX.posAbsolute[2] )
   END_RUNG
   // the same network as SCL:
   #"cathodeAlignTableAxisX Position_"[2](PosiNo := 2,   // "Position.LER_Axis"
                           Status := #unitStatus,
                           int1 := "Unit1.Em5.ControlNodes".cm.softCam.cathodeMainPnP1AxisZ.upPos.inPos,
                           int2 := "Unit1.Em5.ControlNodes".cm.softCam.cathodeMainPnP2AxisZ.upPos.inPos,
                           commands := "Unit1.Em5.HmiInterface".cmCathodeAlignTableAxisX.commands,
                           interlockOk := "Unit1.Em5.ControlNodes".cm.Interlock.cathodeAlignTableAxisX.source.posAbsolute,
                           intOut := "Unit1.Em5.HmiInterface".intCondition.Axis_18.Position.intOut);
   #_w1 := NOT (NOT #FALSE) AND "Unit1.Em5.ControlNodes".cm.Interlock.cathodeAlignTableAxisX.source.posAbsolute[2];
   IF #_w1 THEN "Unit1.Em5.ControlNodes".cmCathodeAlignTableAxisX.commands.selectSetPosition := 2; END_IF;
   "Unit1.Em5.ControlNodes".cm.axisCommand.cathodeAlignTableAxisX.posAbsolute[2] := #_w1;
END_REGION

REGION Network 169: CmCathodeAlignTableAxisX Position Absolute Position3
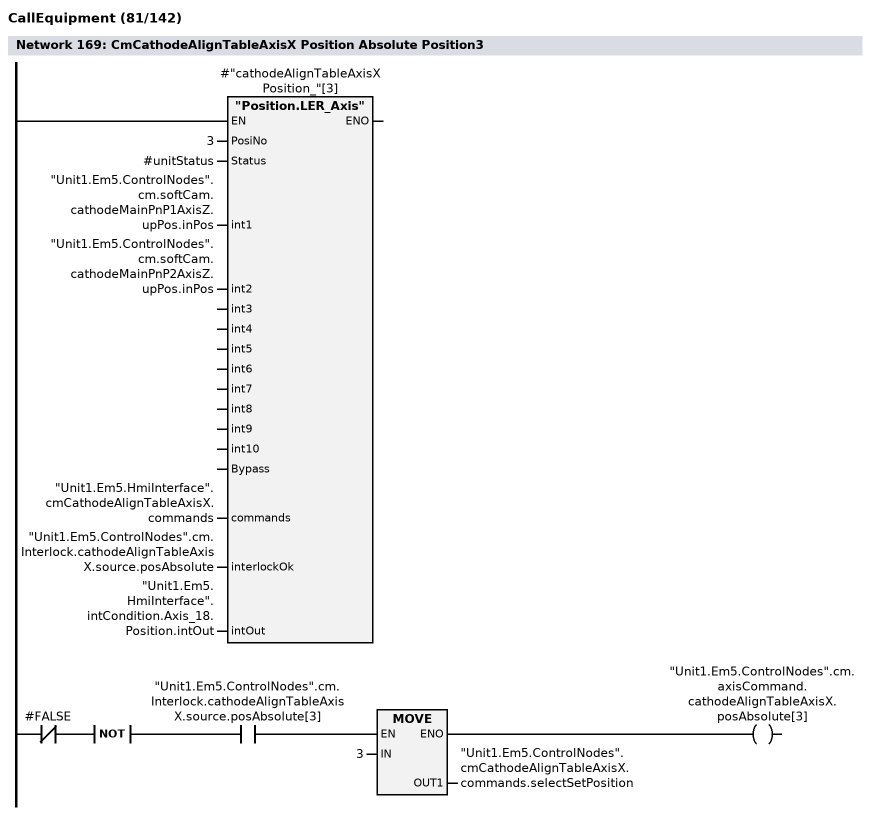
   RUNG wire#powerrail
      #"cathodeAlignTableAxisX Position_"[3](PosiNo := 3, Status := #unitStatus, int1 := "Unit1.Em5.ControlNodes".cm.softCam.cathodeMainPnP1AxisZ.upPos.inPos, int2 := "Unit1.Em5.ControlNodes".cm.softCam.cathodeMainPnP2AxisZ.upPos.inPos, int3 :=, int4 :=, int5 :=, int6 :=, int7 :=, int8 :=, int9 :=, int10 :=, Bypass :=, commands := "Unit1.Em5.HmiInterface".cmCathodeAlignTableAxisX.commands, interlockOk := "Unit1.Em5.ControlNodes".cm.Interlock.cathodeAlignTableAxisX.source.posAbsolute, intOut := "Unit1.Em5.HmiInterface".intCondition.Axis_18.Position.intOut)
   END_RUNG
   RUNG wire#powerrail
      I_Contact( #FALSE )
      Not()
      Contact( "Unit1.Em5.ControlNodes".cm.Interlock.cathodeAlignTableAxisX.source.posAbsolute[3] )
      Move(in := 3, out1 => "Unit1.Em5.ControlNodes".cmCathodeAlignTableAxisX.commands.selectSetPosition)
      Coil( "Unit1.Em5.ControlNodes".cm.axisCommand.cathodeAlignTableAxisX.posAbsolute[3] )
   END_RUNG
   // the same network as SCL:
   #"cathodeAlignTableAxisX Position_"[3](PosiNo := 3,   // "Position.LER_Axis"
                           Status := #unitStatus,
                           int1 := "Unit1.Em5.ControlNodes".cm.softCam.cathodeMainPnP1AxisZ.upPos.inPos,
                           int2 := "Unit1.Em5.ControlNodes".cm.softCam.cathodeMainPnP2AxisZ.upPos.inPos,
                           commands := "Unit1.Em5.HmiInterface".cmCathodeAlignTableAxisX.commands,
                           interlockOk := "Unit1.Em5.ControlNodes".cm.Interlock.cathodeAlignTableAxisX.source.posAbsolute,
                           intOut := "Unit1.Em5.HmiInterface".intCondition.Axis_18.Position.intOut);
   #_w1 := NOT (NOT #FALSE) AND "Unit1.Em5.ControlNodes".cm.Interlock.cathodeAlignTableAxisX.source.posAbsolute[3];
   IF #_w1 THEN "Unit1.Em5.ControlNodes".cmCathodeAlignTableAxisX.commands.selectSetPosition := 3; END_IF;
   "Unit1.Em5.ControlNodes".cm.axisCommand.cathodeAlignTableAxisX.posAbsolute[3] := #_w1;
END_REGION

REGION Network 170: CmCathodeAlignTableAxisX Position Absolute Position4
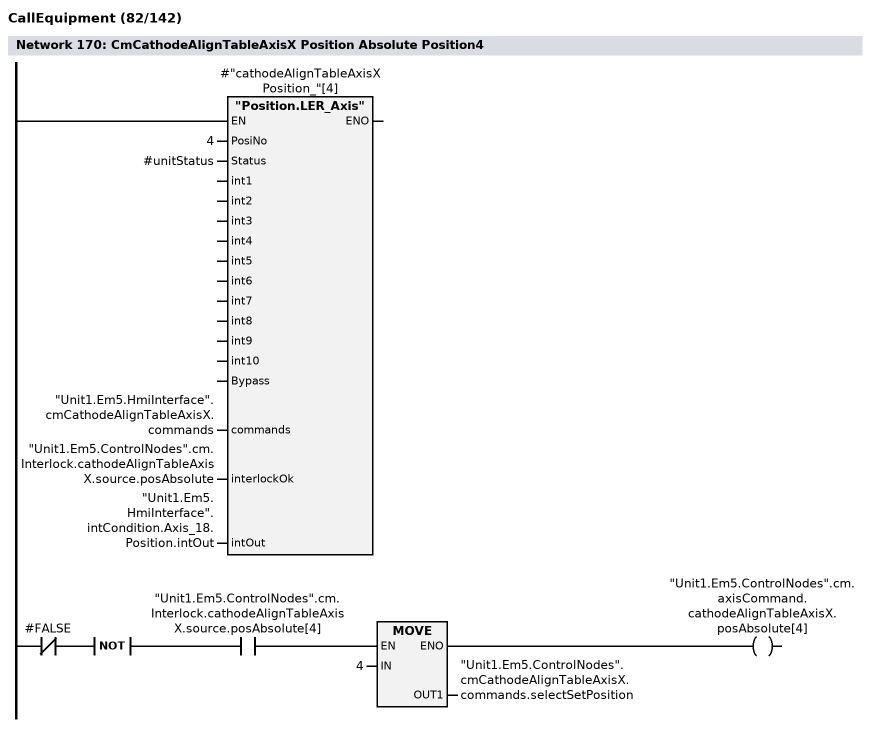
   RUNG wire#powerrail
      #"cathodeAlignTableAxisX Position_"[4](PosiNo := 4, Status := #unitStatus, int1 :=, int2 :=, int3 :=, int4 :=, int5 :=, int6 :=, int7 :=, int8 :=, int9 :=, int10 :=, Bypass :=, commands := "Unit1.Em5.HmiInterface".cmCathodeAlignTableAxisX.commands, interlockOk := "Unit1.Em5.ControlNodes".cm.Interlock.cathodeAlignTableAxisX.source.posAbsolute, intOut := "Unit1.Em5.HmiInterface".intCondition.Axis_18.Position.intOut)
   END_RUNG
   RUNG wire#powerrail
      I_Contact( #FALSE )
      Not()
      Contact( "Unit1.Em5.ControlNodes".cm.Interlock.cathodeAlignTableAxisX.source.posAbsolute[4] )
      Move(in := 4, out1 => "Unit1.Em5.ControlNodes".cmCathodeAlignTableAxisX.commands.selectSetPosition)
      Coil( "Unit1.Em5.ControlNodes".cm.axisCommand.cathodeAlignTableAxisX.posAbsolute[4] )
   END_RUNG
   // the same network as SCL:
   #"cathodeAlignTableAxisX Position_"[4](PosiNo := 4,   // "Position.LER_Axis"
                           Status := #unitStatus,
                           commands := "Unit1.Em5.HmiInterface".cmCathodeAlignTableAxisX.commands,
                           interlockOk := "Unit1.Em5.ControlNodes".cm.Interlock.cathodeAlignTableAxisX.source.posAbsolute,
                           intOut := "Unit1.Em5.HmiInterface".intCondition.Axis_18.Position.intOut);
   #_w1 := NOT (NOT #FALSE) AND "Unit1.Em5.ControlNodes".cm.Interlock.cathodeAlignTableAxisX.source.posAbsolute[4];
   IF #_w1 THEN "Unit1.Em5.ControlNodes".cmCathodeAlignTableAxisX.commands.selectSetPosition := 4; END_IF;
   "Unit1.Em5.ControlNodes".cm.axisCommand.cathodeAlignTableAxisX.posAbsolute[4] := #_w1;
END_REGION

REGION Network 171: CmCathodeAlignTableAxisX Position Absolute Position5
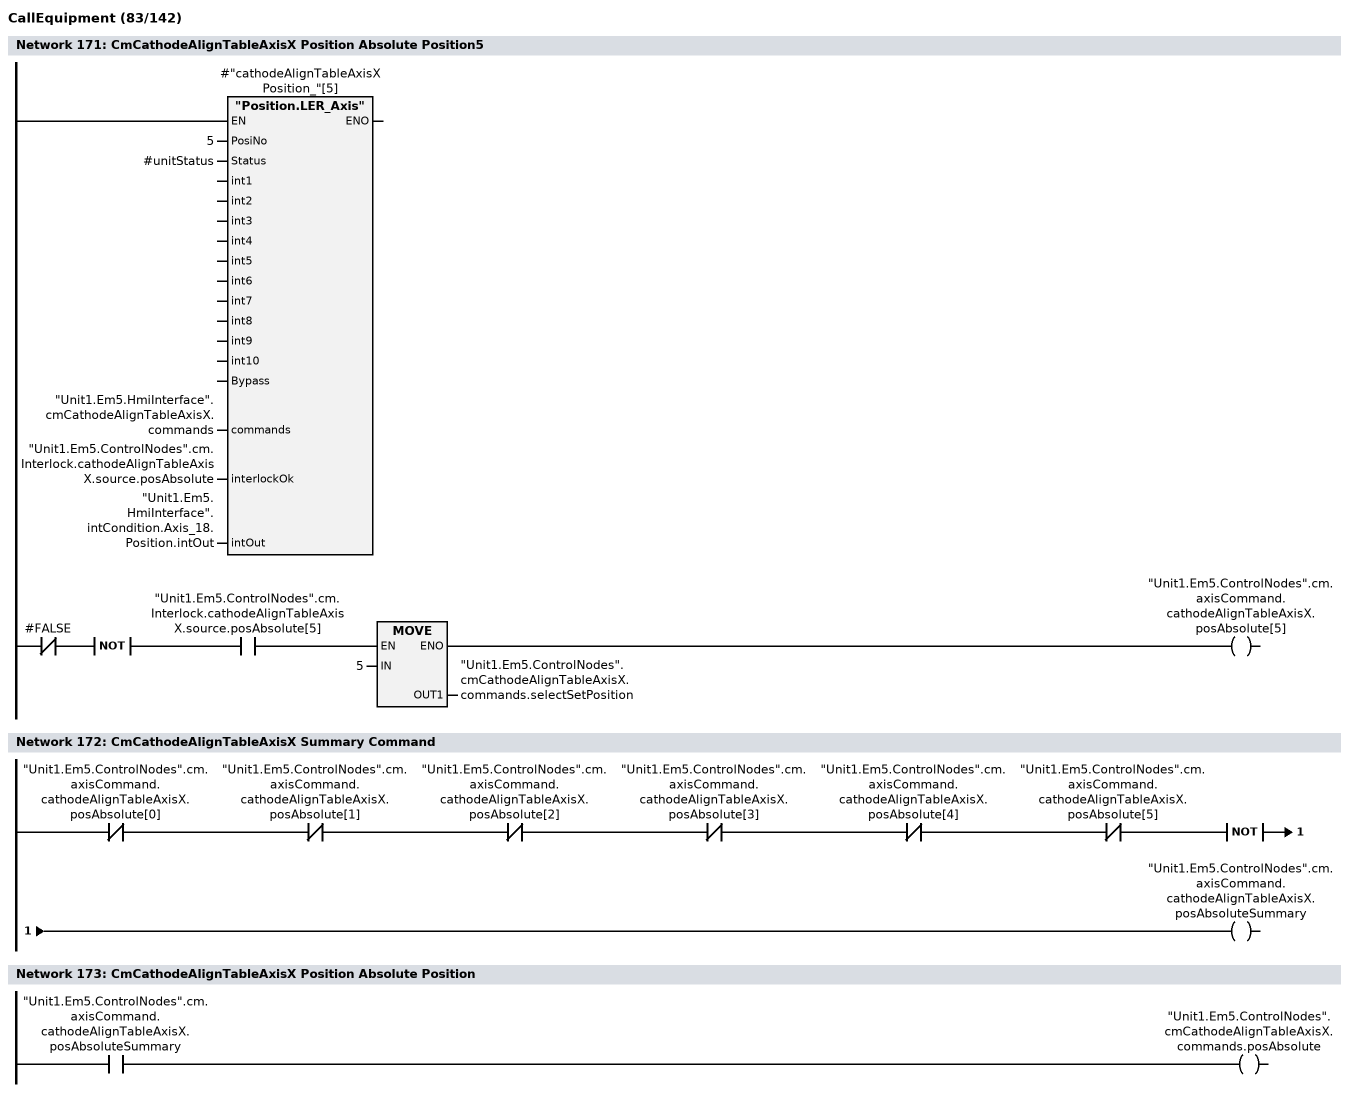
   RUNG wire#powerrail
      #"cathodeAlignTableAxisX Position_"[5](PosiNo := 5, Status := #unitStatus, int1 :=, int2 :=, int3 :=, int4 :=, int5 :=, int6 :=, int7 :=, int8 :=, int9 :=, int10 :=, Bypass :=, commands := "Unit1.Em5.HmiInterface".cmCathodeAlignTableAxisX.commands, interlockOk := "Unit1.Em5.ControlNodes".cm.Interlock.cathodeAlignTableAxisX.source.posAbsolute, intOut := "Unit1.Em5.HmiInterface".intCondition.Axis_18.Position.intOut)
   END_RUNG
   RUNG wire#powerrail
      I_Contact( #FALSE )
      Not()
      Contact( "Unit1.Em5.ControlNodes".cm.Interlock.cathodeAlignTableAxisX.source.posAbsolute[5] )
      Move(in := 5, out1 => "Unit1.Em5.ControlNodes".cmCathodeAlignTableAxisX.commands.selectSetPosition)
      Coil( "Unit1.Em5.ControlNodes".cm.axisCommand.cathodeAlignTableAxisX.posAbsolute[5] )
   END_RUNG
   // the same network as SCL:
   #"cathodeAlignTableAxisX Position_"[5](PosiNo := 5,   // "Position.LER_Axis"
                           Status := #unitStatus,
                           commands := "Unit1.Em5.HmiInterface".cmCathodeAlignTableAxisX.commands,
                           interlockOk := "Unit1.Em5.ControlNodes".cm.Interlock.cathodeAlignTableAxisX.source.posAbsolute,
                           intOut := "Unit1.Em5.HmiInterface".intCondition.Axis_18.Position.intOut);
   #_w1 := NOT (NOT #FALSE) AND "Unit1.Em5.ControlNodes".cm.Interlock.cathodeAlignTableAxisX.source.posAbsolute[5];
   IF #_w1 THEN "Unit1.Em5.ControlNodes".cmCathodeAlignTableAxisX.commands.selectSetPosition := 5; END_IF;
   "Unit1.Em5.ControlNodes".cm.axisCommand.cathodeAlignTableAxisX.posAbsolute[5] := #_w1;
END_REGION

REGION Network 172: CmCathodeAlignTableAxisX Summary Command
   RUNG wire#powerrail
      I_Contact( "Unit1.Em5.ControlNodes".cm.axisCommand.cathodeAlignTableAxisX.posAbsolute[0] )
      I_Contact( "Unit1.Em5.ControlNodes".cm.axisCommand.cathodeAlignTableAxisX.posAbsolute[1] )
      I_Contact( "Unit1.Em5.ControlNodes".cm.axisCommand.cathodeAlignTableAxisX.posAbsolute[2] )
      I_Contact( "Unit1.Em5.ControlNodes".cm.axisCommand.cathodeAlignTableAxisX.posAbsolute[3] )
      I_Contact( "Unit1.Em5.ControlNodes".cm.axisCommand.cathodeAlignTableAxisX.posAbsolute[4] )
      I_Contact( "Unit1.Em5.ControlNodes".cm.axisCommand.cathodeAlignTableAxisX.posAbsolute[5] )
      Not()
      Coil( "Unit1.Em5.ControlNodes".cm.axisCommand.cathodeAlignTableAxisX.posAbsoluteSummary )
   END_RUNG
   // the same network as SCL:
   "Unit1.Em5.ControlNodes".cm.axisCommand.cathodeAlignTableAxisX.posAbsoluteSummary := NOT (NOT "Unit1.Em5.ControlNodes".cm.axisCommand.cathodeAlignTableAxisX.posAbsolute[0] AND NOT "Unit1.Em5.ControlNodes".cm.axisCommand.cathodeAlignTableAxisX.posAbsolute[1] AND NOT "Unit1.Em5.ControlNodes".cm.axisCommand.cathodeAlignTableAxisX.posAbsolute[2] AND NOT "Unit1.Em5.ControlNodes".cm.axisCommand.cathodeAlignTableAxisX.posAbsolute[3] AND NOT "Unit1.Em5.ControlNodes".cm.axisCommand.cathodeAlignTableAxisX.posAbsolute[4] AND NOT "Unit1.Em5.ControlNodes".cm.axisCommand.cathodeAlignTableAxisX.posAbsolute[5]);
END_REGION

REGION Network 173: CmCathodeAlignTableAxisX Position Absolute Position
   RUNG wire#powerrail
      Contact( "Unit1.Em5.ControlNodes".cm.axisCommand.cathodeAlignTableAxisX.posAbsoluteSummary )
      Coil( "Unit1.Em5.ControlNodes".cmCathodeAlignTableAxisX.commands.posAbsolute )
   END_RUNG
   // the same network as SCL:
   "Unit1.Em5.ControlNodes".cmCathodeAlignTableAxisX.commands.posAbsolute := "Unit1.Em5.ControlNodes".cm.axisCommand.cathodeAlignTableAxisX.posAbsoluteSummary;
END_REGION

REGION Network 174: CmCathodeAlignTableAxisX Interlock Summary
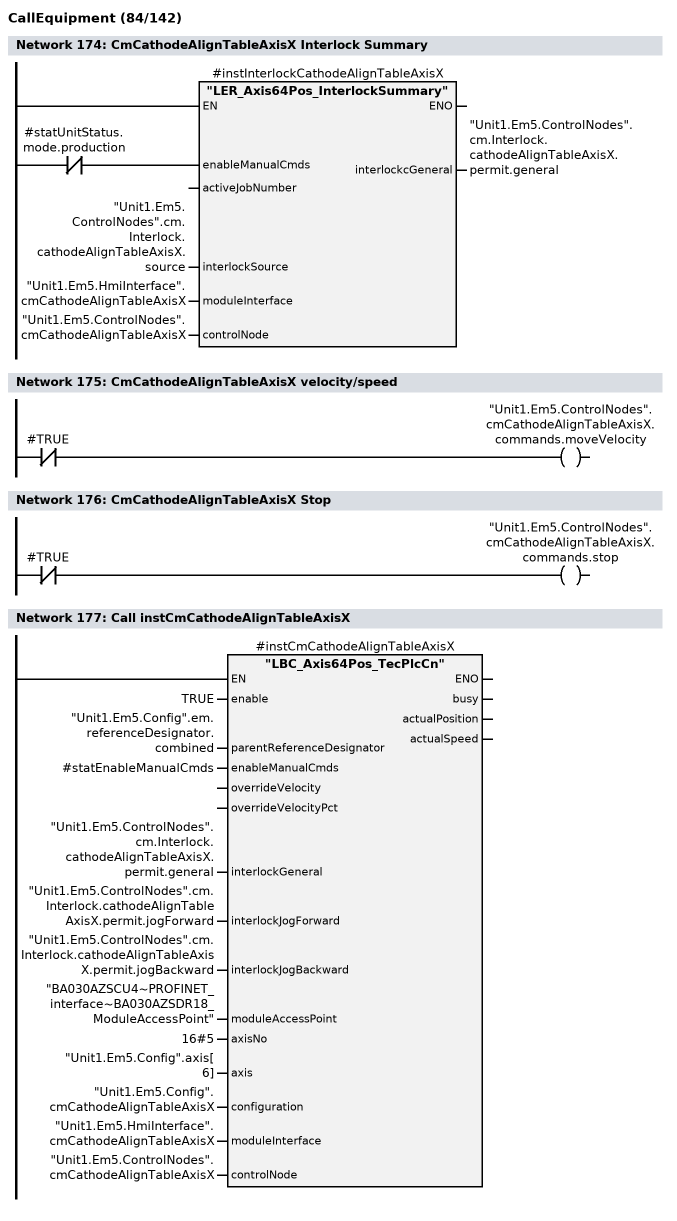
   RUNG wire#powerrail
      #instInterlockCathodeAlignTableAxisX(enableManualCmds := wire#w1, activeJobNumber :=, interlockSource := "Unit1.Em5.ControlNodes".cm.Interlock.cathodeAlignTableAxisX.source, moduleInterface := "Unit1.Em5.HmiInterface".cmCathodeAlignTableAxisX, controlNode := "Unit1.Em5.ControlNodes".cmCathodeAlignTableAxisX, interlockcGeneral => "Unit1.Em5.ControlNodes".cm.Interlock.cathodeAlignTableAxisX.permit.general)
   END_RUNG
   RUNG wire#powerrail
      I_Contact( #statUnitStatus.mode.production )
   END_RUNG wire#w1
   // the same network as SCL:
   #instInterlockCathodeAlignTableAxisX(enableManualCmds := NOT #statUnitStatus.mode.production,   // "LER_Axis64Pos_InterlockSummary"
                           interlockSource := "Unit1.Em5.ControlNodes".cm.Interlock.cathodeAlignTableAxisX.source,
                           moduleInterface := "Unit1.Em5.HmiInterface".cmCathodeAlignTableAxisX,
                           controlNode := "Unit1.Em5.ControlNodes".cmCathodeAlignTableAxisX,
                           interlockcGeneral => "Unit1.Em5.ControlNodes".cm.Interlock.cathodeAlignTableAxisX.permit.general);
END_REGION

REGION Network 175: CmCathodeAlignTableAxisX velocity/speed
   RUNG wire#powerrail
      I_Contact( #TRUE )
      Coil( "Unit1.Em5.ControlNodes".cmCathodeAlignTableAxisX.commands.moveVelocity )
   END_RUNG
   // the same network as SCL:
   "Unit1.Em5.ControlNodes".cmCathodeAlignTableAxisX.commands.moveVelocity := NOT #TRUE;
END_REGION

REGION Network 176: CmCathodeAlignTableAxisX Stop
   RUNG wire#powerrail
      I_Contact( #TRUE )
      Coil( "Unit1.Em5.ControlNodes".cmCathodeAlignTableAxisX.commands.stop )
   END_RUNG
   // the same network as SCL:
   "Unit1.Em5.ControlNodes".cmCathodeAlignTableAxisX.commands.stop := NOT #TRUE;
END_REGION

REGION Network 177: Call instCmCathodeAlignTableAxisX
   RUNG wire#powerrail
      #instCmCathodeAlignTableAxisX(enable := TRUE, parentReferenceDesignator := "Unit1.Em5.Config".em.referenceDesignator.combined, enableManualCmds := #statEnableManualCmds, overrideVelocity :=, overrideVelocityPct :=, interlockGeneral := "Unit1.Em5.ControlNodes".cm.Interlock.cathodeAlignTableAxisX.permit.general, interlockJogForward := "Unit1.Em5.ControlNodes".cm.Interlock.cathodeAlignTableAxisX.permit.jogForward, interlockJogBackward := "Unit1.Em5.ControlNodes".cm.Interlock.cathodeAlignTableAxisX.permit.jogBackward, moduleAccessPoint := "BA030AZSCU4~PROFINET_interface~BA030AZSDR18_ModuleAccessPoint", axisNo := 16#5, axis := "Unit1.Em5.Config".axis[6], configuration := "Unit1.Em5.Config".cmCathodeAlignTableAxisX, moduleInterface := "Unit1.Em5.HmiInterface".cmCathodeAlignTableAxisX, controlNode := "Unit1.Em5.ControlNodes".cmCathodeAlignTableAxisX, busy =>, actualPosition =>, actualSpeed =>)
   END_RUNG
   // the same network as SCL:
   #instCmCathodeAlignTableAxisX(enable := TRUE,   // "LBC_Axis64Pos_TecPlcCn"
                           parentReferenceDesignator := "Unit1.Em5.Config".em.referenceDesignator.combined,
                           enableManualCmds := #statEnableManualCmds,
                           interlockGeneral := "Unit1.Em5.ControlNodes".cm.Interlock.cathodeAlignTableAxisX.permit.general,
                           interlockJogForward := "Unit1.Em5.ControlNodes".cm.Interlock.cathodeAlignTableAxisX.permit.jogForward,
                           interlockJogBackward := "Unit1.Em5.ControlNodes".cm.Interlock.cathodeAlignTableAxisX.permit.jogBackward,
                           moduleAccessPoint := "BA030AZSCU4~PROFINET_interface~BA030AZSDR18_ModuleAccessPoint",
                           axisNo := 16#5,
                           axis := "Unit1.Em5.Config".axis[6],
                           configuration := "Unit1.Em5.Config".cmCathodeAlignTableAxisX,
                           moduleInterface := "Unit1.Em5.HmiInterface".cmCathodeAlignTableAxisX,
                           controlNode := "Unit1.Em5.ControlNodes".cmCathodeAlignTableAxisX);
END_REGION

REGION Network 178: CmCathodeAlignTableAxisX SoftCam
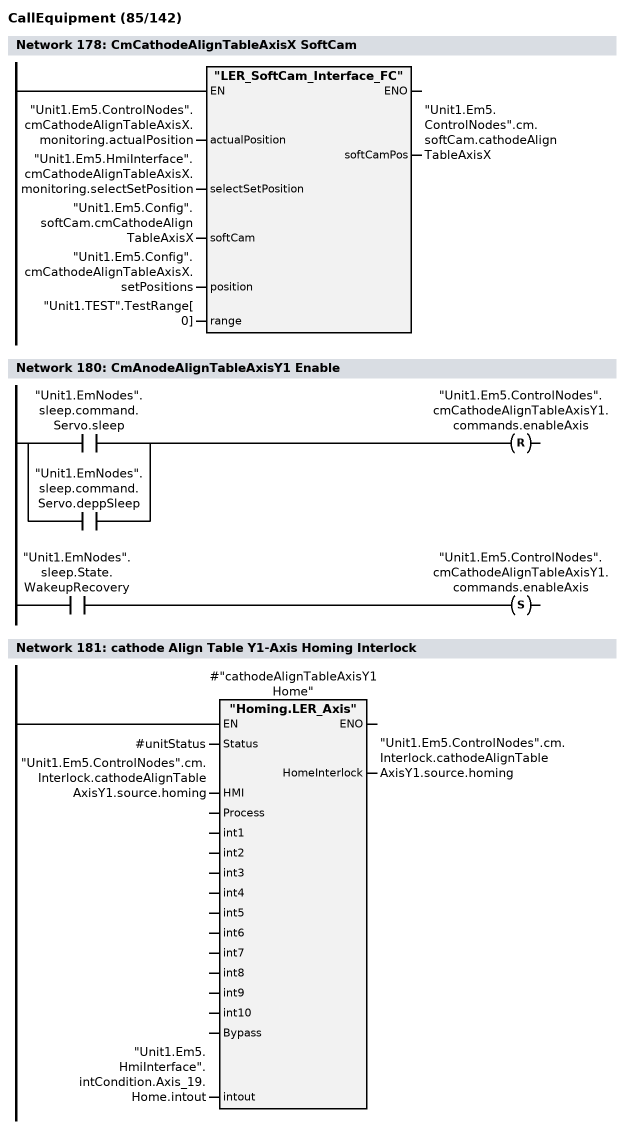
   RUNG wire#powerrail
      "LER_SoftCam_Interface_FC"(actualPosition := "Unit1.Em5.ControlNodes".cmCathodeAlignTableAxisX.monitoring.actualPosition, selectSetPosition := "Unit1.Em5.HmiInterface".cmCathodeAlignTableAxisX.monitoring.selectSetPosition, softCam := "Unit1.Em5.Config".softCam.cmCathodeAlignTableAxisX, position := "Unit1.Em5.Config".cmCathodeAlignTableAxisX.setPositions, range := "Unit1.TEST".TestRange[0], softCamPos => "Unit1.Em5.ControlNodes".cm.softCam.cathodeAlignTableAxisX)
   END_RUNG
   // the same network as SCL:
   "LER_SoftCam_Interface_FC"(actualPosition := "Unit1.Em5.ControlNodes".cmCathodeAlignTableAxisX.monitoring.actualPosition,
                           selectSetPosition := "Unit1.Em5.HmiInterface".cmCathodeAlignTableAxisX.monitoring.selectSetPosition,
                           softCam := "Unit1.Em5.Config".softCam.cmCathodeAlignTableAxisX,
                           position := "Unit1.Em5.Config".cmCathodeAlignTableAxisX.setPositions,
                           range := "Unit1.TEST".TestRange[0],
                           softCamPos => "Unit1.Em5.ControlNodes".cm.softCam.cathodeAlignTableAxisX);
END_REGION

REGION Network 180: CmAnodeAlignTableAxisY1 Enable
   RUNG wire#powerrail
      Contact( "Unit1.EmNodes".sleep.command.Servo.sleep )
      wire#w1
      R_Coil( "Unit1.Em5.ControlNodes".cmCathodeAlignTableAxisY1.commands.enableAxis )
   END_RUNG
   RUNG wire#powerrail
      Contact( "Unit1.EmNodes".sleep.command.Servo.deppSleep )
   END_RUNG wire#w1
   RUNG wire#powerrail
      Contact( "Unit1.EmNodes".sleep.State.WakeupRecovery )
      S_Coil( "Unit1.Em5.ControlNodes".cmCathodeAlignTableAxisY1.commands.enableAxis )
   END_RUNG
   // the same network as SCL:
   IF "Unit1.EmNodes".sleep.command.Servo.sleep OR "Unit1.EmNodes".sleep.command.Servo.deppSleep THEN
       "Unit1.Em5.ControlNodes".cmCathodeAlignTableAxisY1.commands.enableAxis := FALSE;
   END_IF;
   IF "Unit1.EmNodes".sleep.State.WakeupRecovery THEN
       "Unit1.Em5.ControlNodes".cmCathodeAlignTableAxisY1.commands.enableAxis := TRUE;
   END_IF;
END_REGION

REGION Network 181: cathode Align Table Y1-Axis Homing Interlock
   RUNG wire#powerrail
      #"cathodeAlignTableAxisY1 Home"(Status := #unitStatus, HMI := "Unit1.Em5.ControlNodes".cm.Interlock.cathodeAlignTableAxisY1.source.homing, Process :=, int1 :=, int2 :=, int3 :=, int4 :=, int5 :=, int6 :=, int7 :=, int8 :=, int9 :=, int10 :=, Bypass :=, intout := "Unit1.Em5.HmiInterface".intCondition.Axis_19.Home.intout, HomeInterlock => "Unit1.Em5.ControlNodes".cm.Interlock.cathodeAlignTableAxisY1.source.homing)
   END_RUNG
   // the same network as SCL:
   #"cathodeAlignTableAxisY1 Home"(Status := #unitStatus,   // "Homing.LER_Axis"
                           HMI := "Unit1.Em5.ControlNodes".cm.Interlock.cathodeAlignTableAxisY1.source.homing,
                           intout := "Unit1.Em5.HmiInterface".intCondition.Axis_19.Home.intout,
                           HomeInterlock => "Unit1.Em5.ControlNodes".cm.Interlock.cathodeAlignTableAxisY1.source.homing);
END_REGION

REGION Network 182: CmCathodeAlignTableAxisY1 Position Absolute Jog
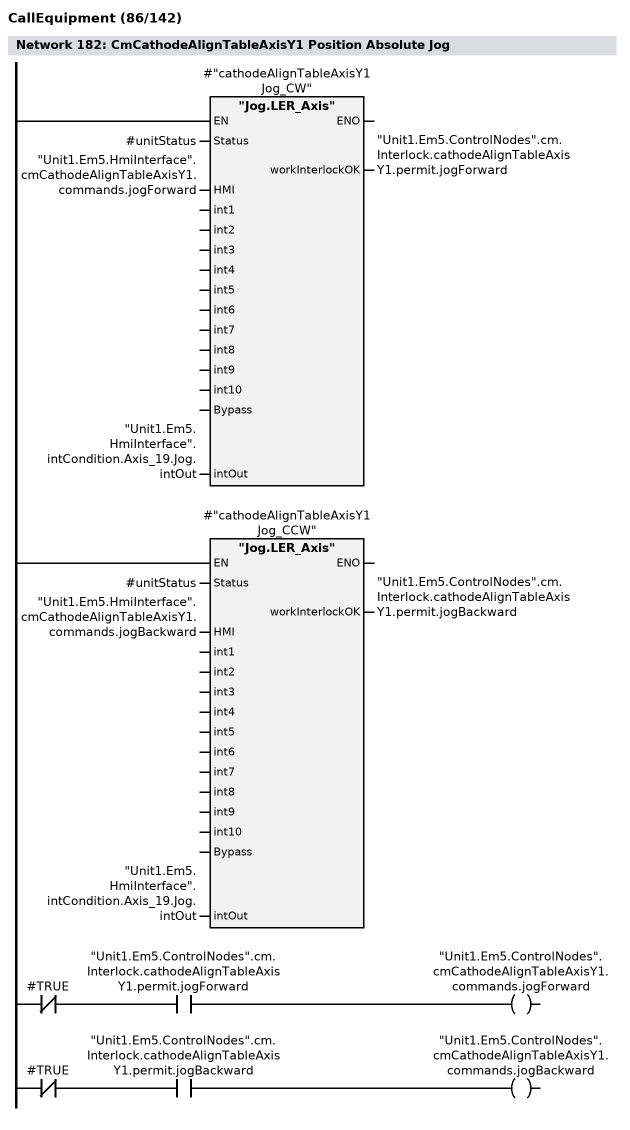
   RUNG wire#powerrail
      #"cathodeAlignTableAxisY1 Jog_CW"(Status := #unitStatus, HMI := "Unit1.Em5.HmiInterface".cmCathodeAlignTableAxisY1.commands.jogForward, int1 :=, int2 :=, int3 :=, int4 :=, int5 :=, int6 :=, int7 :=, int8 :=, int9 :=, int10 :=, Bypass :=, intOut := "Unit1.Em5.HmiInterface".intCondition.Axis_19.Jog.intOut, workInterlockOK => "Unit1.Em5.ControlNodes".cm.Interlock.cathodeAlignTableAxisY1.permit.jogForward)
   END_RUNG
   RUNG wire#powerrail
      #"cathodeAlignTableAxisY1 Jog_CCW"(Status := #unitStatus, HMI := "Unit1.Em5.HmiInterface".cmCathodeAlignTableAxisY1.commands.jogBackward, int1 :=, int2 :=, int3 :=, int4 :=, int5 :=, int6 :=, int7 :=, int8 :=, int9 :=, int10 :=, Bypass :=, intOut := "Unit1.Em5.HmiInterface".intCondition.Axis_19.Jog.intOut, workInterlockOK => "Unit1.Em5.ControlNodes".cm.Interlock.cathodeAlignTableAxisY1.permit.jogBackward)
   END_RUNG
   RUNG wire#powerrail
      I_Contact( #TRUE )
      Contact( "Unit1.Em5.ControlNodes".cm.Interlock.cathodeAlignTableAxisY1.permit.jogForward )
      Coil( "Unit1.Em5.ControlNodes".cmCathodeAlignTableAxisY1.commands.jogForward )
   END_RUNG
   RUNG wire#powerrail
      I_Contact( #TRUE )
      Contact( "Unit1.Em5.ControlNodes".cm.Interlock.cathodeAlignTableAxisY1.permit.jogBackward )
      Coil( "Unit1.Em5.ControlNodes".cmCathodeAlignTableAxisY1.commands.jogBackward )
   END_RUNG
   // the same network as SCL:
   #"cathodeAlignTableAxisY1 Jog_CW"(Status := #unitStatus,   // "Jog.LER_Axis"
                           HMI := "Unit1.Em5.HmiInterface".cmCathodeAlignTableAxisY1.commands.jogForward,
                           intOut := "Unit1.Em5.HmiInterface".intCondition.Axis_19.Jog.intOut,
                           workInterlockOK => "Unit1.Em5.ControlNodes".cm.Interlock.cathodeAlignTableAxisY1.permit.jogForward);
   #"cathodeAlignTableAxisY1 Jog_CCW"(Status := #unitStatus,   // "Jog.LER_Axis"
                           HMI := "Unit1.Em5.HmiInterface".cmCathodeAlignTableAxisY1.commands.jogBackward,
                           intOut := "Unit1.Em5.HmiInterface".intCondition.Axis_19.Jog.intOut,
                           workInterlockOK => "Unit1.Em5.ControlNodes".cm.Interlock.cathodeAlignTableAxisY1.permit.jogBackward);
   "Unit1.Em5.ControlNodes".cmCathodeAlignTableAxisY1.commands.jogForward := NOT #TRUE AND "Unit1.Em5.ControlNodes".cm.Interlock.cathodeAlignTableAxisY1.permit.jogForward;
   "Unit1.Em5.ControlNodes".cmCathodeAlignTableAxisY1.commands.jogBackward := NOT #TRUE AND "Unit1.Em5.ControlNodes".cm.Interlock.cathodeAlignTableAxisY1.permit.jogBackward;
END_REGION

REGION Network 183: CmCathodeAlignTableAxisY1 Position Absolute Position0
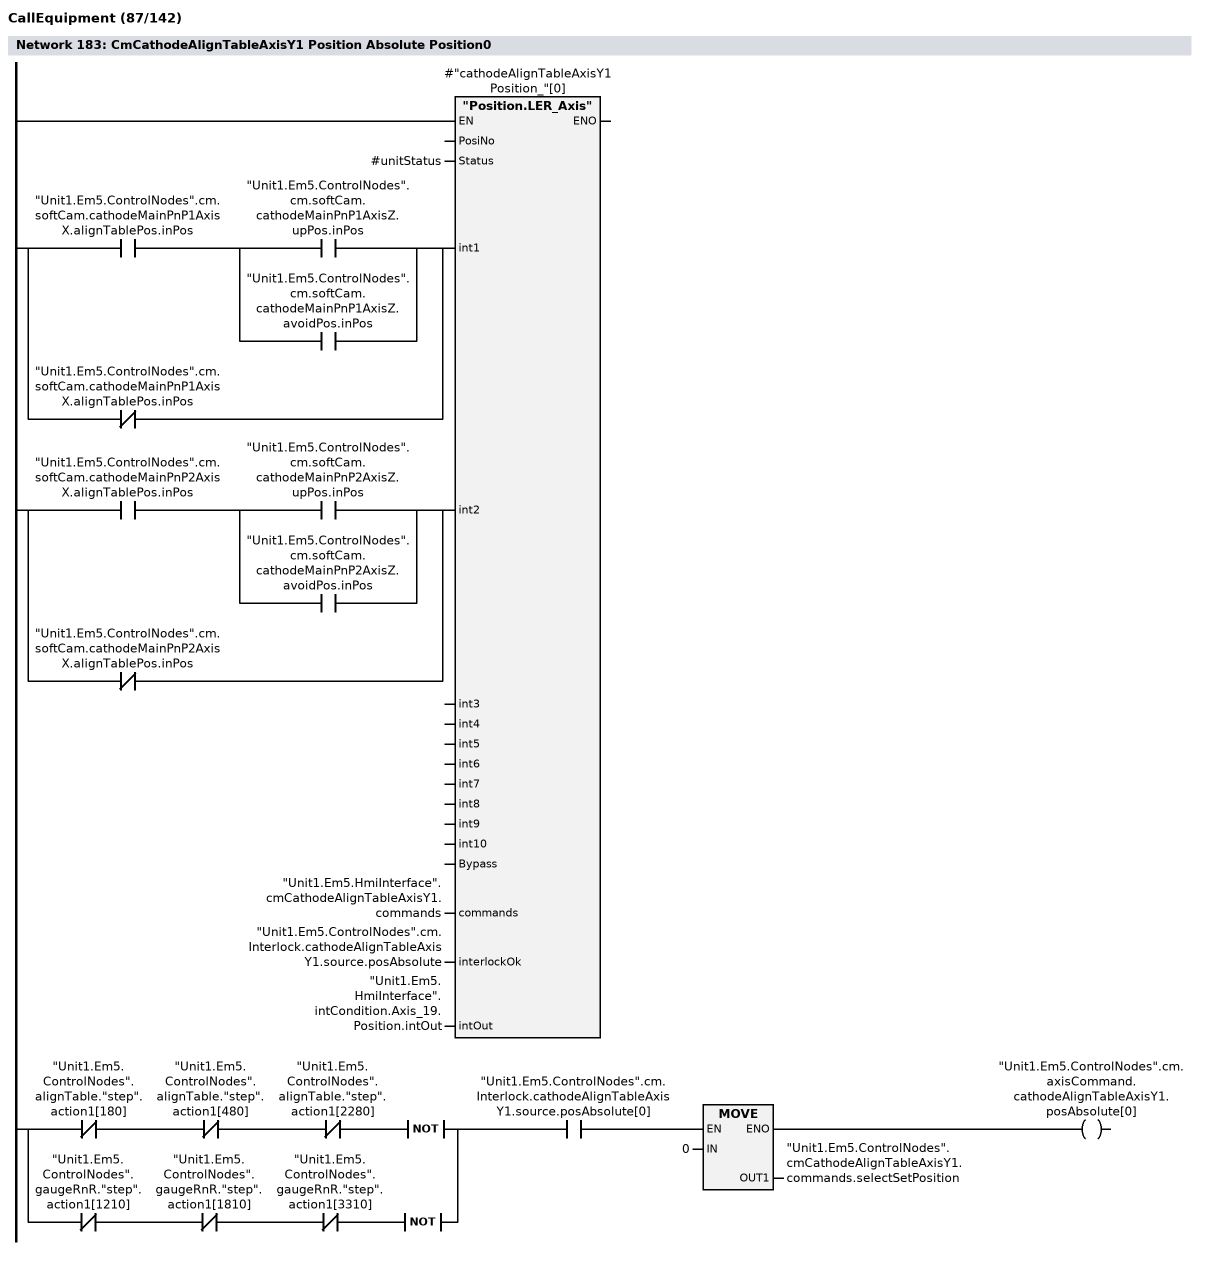
   RUNG wire#powerrail
      #"cathodeAlignTableAxisY1 Position_"[0](int1 := wire#w2, int2 := wire#w4, PosiNo :=, Status := #unitStatus, int3 :=, int4 :=, int5 :=, int6 :=, int7 :=, int8 :=, int9 :=, int10 :=, Bypass :=, commands := "Unit1.Em5.HmiInterface".cmCathodeAlignTableAxisY1.commands, interlockOk := "Unit1.Em5.ControlNodes".cm.Interlock.cathodeAlignTableAxisY1.source.posAbsolute, intOut := "Unit1.Em5.HmiInterface".intCondition.Axis_19.Position.intOut)
   END_RUNG
   RUNG wire#powerrail
      Contact( "Unit1.Em5.ControlNodes".cm.softCam.cathodeMainPnP1AxisX.alignTablePos.inPos )
      wire#w1
      Contact( "Unit1.Em5.ControlNodes".cm.softCam.cathodeMainPnP1AxisZ.upPos.inPos )
   END_RUNG wire#w2
   RUNG wire#w1
      Contact( "Unit1.Em5.ControlNodes".cm.softCam.cathodeMainPnP1AxisZ.avoidPos.inPos )
   END_RUNG wire#w2
   RUNG wire#powerrail
      I_Contact( "Unit1.Em5.ControlNodes".cm.softCam.cathodeMainPnP1AxisX.alignTablePos.inPos )
   END_RUNG wire#w2
   RUNG wire#powerrail
      Contact( "Unit1.Em5.ControlNodes".cm.softCam.cathodeMainPnP2AxisX.alignTablePos.inPos )
      wire#w3
      Contact( "Unit1.Em5.ControlNodes".cm.softCam.cathodeMainPnP2AxisZ.upPos.inPos )
   END_RUNG wire#w4
   RUNG wire#w3
      Contact( "Unit1.Em5.ControlNodes".cm.softCam.cathodeMainPnP2AxisZ.avoidPos.inPos )
   END_RUNG wire#w4
   RUNG wire#powerrail
      I_Contact( "Unit1.Em5.ControlNodes".cm.softCam.cathodeMainPnP2AxisX.alignTablePos.inPos )
   END_RUNG wire#w4
   RUNG wire#powerrail
      I_Contact( "Unit1.Em5.ControlNodes".alignTable."step".action1[180] )
      I_Contact( "Unit1.Em5.ControlNodes".alignTable."step".action1[480] )
      I_Contact( "Unit1.Em5.ControlNodes".alignTable."step".action1[2280] )
      Not()
      wire#w5
      Contact( "Unit1.Em5.ControlNodes".cm.Interlock.cathodeAlignTableAxisY1.source.posAbsolute[0] )
      Move(in := 0, out1 => "Unit1.Em5.ControlNodes".cmCathodeAlignTableAxisY1.commands.selectSetPosition)
      Coil( "Unit1.Em5.ControlNodes".cm.axisCommand.cathodeAlignTableAxisY1.posAbsolute[0] )
   END_RUNG
   RUNG wire#powerrail
      I_Contact( "Unit1.Em5.ControlNodes".gaugeRnR."step".action1[1210] )
      I_Contact( "Unit1.Em5.ControlNodes".gaugeRnR."step".action1[1810] )
      I_Contact( "Unit1.Em5.ControlNodes".gaugeRnR."step".action1[3310] )
      Not()
   END_RUNG wire#w5
   // the same network as SCL:
   #"cathodeAlignTableAxisY1 Position_"[0](Status := #unitStatus,   // "Position.LER_Axis"
                           int1 := ("Unit1.Em5.ControlNodes".cm.softCam.cathodeMainPnP1AxisX.alignTablePos.inPos AND ("Unit1.Em5.ControlNodes".cm.softCam.cathodeMainPnP1AxisZ.upPos.inPos OR "Unit1.Em5.ControlNodes".cm.softCam.cathodeMainPnP1AxisZ.avoidPos.inPos)) OR NOT "Unit1.Em5.ControlNodes".cm.softCam.cathodeMainPnP1AxisX.alignTablePos.inPos,
                           int2 := ("Unit1.Em5.ControlNodes".cm.softCam.cathodeMainPnP2AxisX.alignTablePos.inPos AND ("Unit1.Em5.ControlNodes".cm.softCam.cathodeMainPnP2AxisZ.upPos.inPos OR "Unit1.Em5.ControlNodes".cm.softCam.cathodeMainPnP2AxisZ.avoidPos.inPos)) OR NOT "Unit1.Em5.ControlNodes".cm.softCam.cathodeMainPnP2AxisX.alignTablePos.inPos,
                           commands := "Unit1.Em5.HmiInterface".cmCathodeAlignTableAxisY1.commands,
                           interlockOk := "Unit1.Em5.ControlNodes".cm.Interlock.cathodeAlignTableAxisY1.source.posAbsolute,
                           intOut := "Unit1.Em5.HmiInterface".intCondition.Axis_19.Position.intOut);
   #_w1 := (NOT (NOT "Unit1.Em5.ControlNodes".alignTable."step".action1[180] AND NOT "Unit1.Em5.ControlNodes".alignTable."step".action1[480] AND NOT "Unit1.Em5.ControlNodes".alignTable."step".action1[2280]) OR NOT (NOT "Unit1.Em5.ControlNodes".gaugeRnR."step".action1[1210] AND NOT "Unit1.Em5.ControlNodes".gaugeRnR."step".action1[1810] AND NOT "Unit1.Em5.ControlNodes".gaugeRnR."step".action1[3310])) AND "Unit1.Em5.ControlNodes".cm.Interlock.cathodeAlignTableAxisY1.source.posAbsolute[0];
   IF #_w1 THEN "Unit1.Em5.ControlNodes".cmCathodeAlignTableAxisY1.commands.selectSetPosition := 0; END_IF;
   "Unit1.Em5.ControlNodes".cm.axisCommand.cathodeAlignTableAxisY1.posAbsolute[0] := #_w1;
END_REGION

REGION Network 184: CmCathodeAlignTableAxisY1 Position Absolute Position1
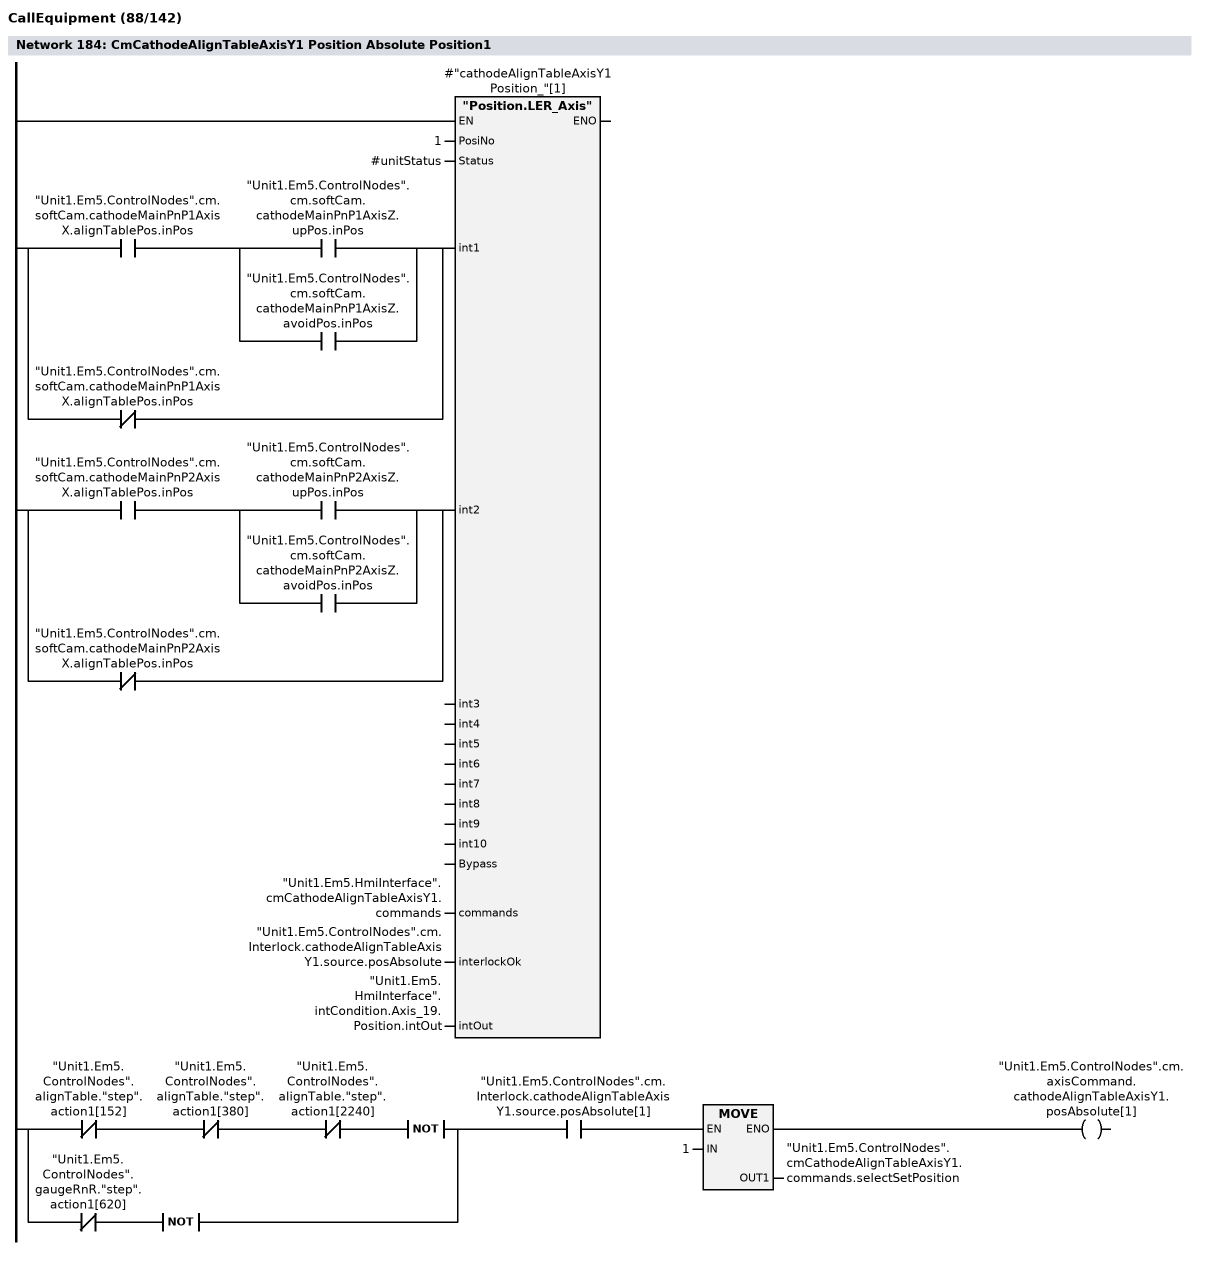
   RUNG wire#powerrail
      #"cathodeAlignTableAxisY1 Position_"[1](int1 := wire#w2, int2 := wire#w4, PosiNo := 1, Status := #unitStatus, int3 :=, int4 :=, int5 :=, int6 :=, int7 :=, int8 :=, int9 :=, int10 :=, Bypass :=, commands := "Unit1.Em5.HmiInterface".cmCathodeAlignTableAxisY1.commands, interlockOk := "Unit1.Em5.ControlNodes".cm.Interlock.cathodeAlignTableAxisY1.source.posAbsolute, intOut := "Unit1.Em5.HmiInterface".intCondition.Axis_19.Position.intOut)
   END_RUNG
   RUNG wire#powerrail
      Contact( "Unit1.Em5.ControlNodes".cm.softCam.cathodeMainPnP1AxisX.alignTablePos.inPos )
      wire#w1
      Contact( "Unit1.Em5.ControlNodes".cm.softCam.cathodeMainPnP1AxisZ.upPos.inPos )
   END_RUNG wire#w2
   RUNG wire#w1
      Contact( "Unit1.Em5.ControlNodes".cm.softCam.cathodeMainPnP1AxisZ.avoidPos.inPos )
   END_RUNG wire#w2
   RUNG wire#powerrail
      I_Contact( "Unit1.Em5.ControlNodes".cm.softCam.cathodeMainPnP1AxisX.alignTablePos.inPos )
   END_RUNG wire#w2
   RUNG wire#powerrail
      Contact( "Unit1.Em5.ControlNodes".cm.softCam.cathodeMainPnP2AxisX.alignTablePos.inPos )
      wire#w3
      Contact( "Unit1.Em5.ControlNodes".cm.softCam.cathodeMainPnP2AxisZ.upPos.inPos )
   END_RUNG wire#w4
   RUNG wire#w3
      Contact( "Unit1.Em5.ControlNodes".cm.softCam.cathodeMainPnP2AxisZ.avoidPos.inPos )
   END_RUNG wire#w4
   RUNG wire#powerrail
      I_Contact( "Unit1.Em5.ControlNodes".cm.softCam.cathodeMainPnP2AxisX.alignTablePos.inPos )
   END_RUNG wire#w4
   RUNG wire#powerrail
      I_Contact( "Unit1.Em5.ControlNodes".alignTable."step".action1[152] )
      I_Contact( "Unit1.Em5.ControlNodes".alignTable."step".action1[380] )
      I_Contact( "Unit1.Em5.ControlNodes".alignTable."step".action1[2240] )
      Not()
      wire#w5
      Contact( "Unit1.Em5.ControlNodes".cm.Interlock.cathodeAlignTableAxisY1.source.posAbsolute[1] )
      Move(in := 1, out1 => "Unit1.Em5.ControlNodes".cmCathodeAlignTableAxisY1.commands.selectSetPosition)
      Coil( "Unit1.Em5.ControlNodes".cm.axisCommand.cathodeAlignTableAxisY1.posAbsolute[1] )
   END_RUNG
   RUNG wire#powerrail
      I_Contact( "Unit1.Em5.ControlNodes".gaugeRnR."step".action1[620] )
      Not()
   END_RUNG wire#w5
   // the same network as SCL:
   #"cathodeAlignTableAxisY1 Position_"[1](PosiNo := 1,   // "Position.LER_Axis"
                           Status := #unitStatus,
                           int1 := ("Unit1.Em5.ControlNodes".cm.softCam.cathodeMainPnP1AxisX.alignTablePos.inPos AND ("Unit1.Em5.ControlNodes".cm.softCam.cathodeMainPnP1AxisZ.upPos.inPos OR "Unit1.Em5.ControlNodes".cm.softCam.cathodeMainPnP1AxisZ.avoidPos.inPos)) OR NOT "Unit1.Em5.ControlNodes".cm.softCam.cathodeMainPnP1AxisX.alignTablePos.inPos,
                           int2 := ("Unit1.Em5.ControlNodes".cm.softCam.cathodeMainPnP2AxisX.alignTablePos.inPos AND ("Unit1.Em5.ControlNodes".cm.softCam.cathodeMainPnP2AxisZ.upPos.inPos OR "Unit1.Em5.ControlNodes".cm.softCam.cathodeMainPnP2AxisZ.avoidPos.inPos)) OR NOT "Unit1.Em5.ControlNodes".cm.softCam.cathodeMainPnP2AxisX.alignTablePos.inPos,
                           commands := "Unit1.Em5.HmiInterface".cmCathodeAlignTableAxisY1.commands,
                           interlockOk := "Unit1.Em5.ControlNodes".cm.Interlock.cathodeAlignTableAxisY1.source.posAbsolute,
                           intOut := "Unit1.Em5.HmiInterface".intCondition.Axis_19.Position.intOut);
   #_w1 := (NOT (NOT "Unit1.Em5.ControlNodes".alignTable."step".action1[152] AND NOT "Unit1.Em5.ControlNodes".alignTable."step".action1[380] AND NOT "Unit1.Em5.ControlNodes".alignTable."step".action1[2240]) OR NOT (NOT "Unit1.Em5.ControlNodes".gaugeRnR."step".action1[620])) AND "Unit1.Em5.ControlNodes".cm.Interlock.cathodeAlignTableAxisY1.source.posAbsolute[1];
   IF #_w1 THEN "Unit1.Em5.ControlNodes".cmCathodeAlignTableAxisY1.commands.selectSetPosition := 1; END_IF;
   "Unit1.Em5.ControlNodes".cm.axisCommand.cathodeAlignTableAxisY1.posAbsolute[1] := #_w1;
END_REGION

REGION Network 185: CmCathodeAlignTableAxisY1 Position Absolute Position2
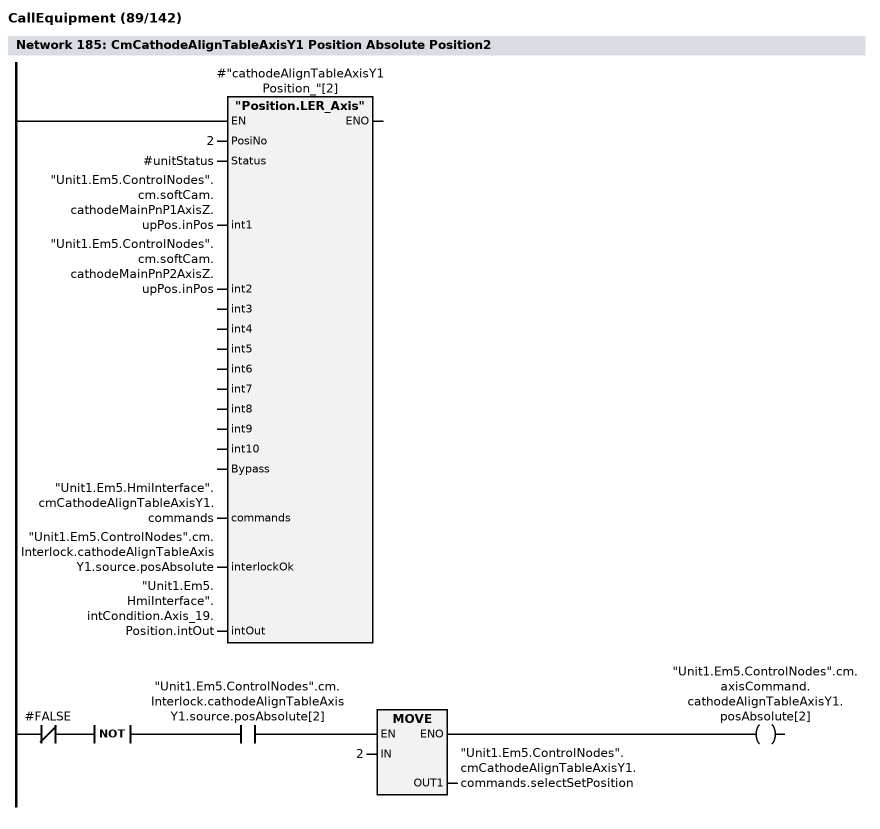
   RUNG wire#powerrail
      #"cathodeAlignTableAxisY1 Position_"[2](PosiNo := 2, Status := #unitStatus, int1 := "Unit1.Em5.ControlNodes".cm.softCam.cathodeMainPnP1AxisZ.upPos.inPos, int2 := "Unit1.Em5.ControlNodes".cm.softCam.cathodeMainPnP2AxisZ.upPos.inPos, int3 :=, int4 :=, int5 :=, int6 :=, int7 :=, int8 :=, int9 :=, int10 :=, Bypass :=, commands := "Unit1.Em5.HmiInterface".cmCathodeAlignTableAxisY1.commands, interlockOk := "Unit1.Em5.ControlNodes".cm.Interlock.cathodeAlignTableAxisY1.source.posAbsolute, intOut := "Unit1.Em5.HmiInterface".intCondition.Axis_19.Position.intOut)
   END_RUNG
   RUNG wire#powerrail
      I_Contact( #FALSE )
      Not()
      Contact( "Unit1.Em5.ControlNodes".cm.Interlock.cathodeAlignTableAxisY1.source.posAbsolute[2] )
      Move(in := 2, out1 => "Unit1.Em5.ControlNodes".cmCathodeAlignTableAxisY1.commands.selectSetPosition)
      Coil( "Unit1.Em5.ControlNodes".cm.axisCommand.cathodeAlignTableAxisY1.posAbsolute[2] )
   END_RUNG
   // the same network as SCL:
   #"cathodeAlignTableAxisY1 Position_"[2](PosiNo := 2,   // "Position.LER_Axis"
                           Status := #unitStatus,
                           int1 := "Unit1.Em5.ControlNodes".cm.softCam.cathodeMainPnP1AxisZ.upPos.inPos,
                           int2 := "Unit1.Em5.ControlNodes".cm.softCam.cathodeMainPnP2AxisZ.upPos.inPos,
                           commands := "Unit1.Em5.HmiInterface".cmCathodeAlignTableAxisY1.commands,
                           interlockOk := "Unit1.Em5.ControlNodes".cm.Interlock.cathodeAlignTableAxisY1.source.posAbsolute,
                           intOut := "Unit1.Em5.HmiInterface".intCondition.Axis_19.Position.intOut);
   #_w1 := NOT (NOT #FALSE) AND "Unit1.Em5.ControlNodes".cm.Interlock.cathodeAlignTableAxisY1.source.posAbsolute[2];
   IF #_w1 THEN "Unit1.Em5.ControlNodes".cmCathodeAlignTableAxisY1.commands.selectSetPosition := 2; END_IF;
   "Unit1.Em5.ControlNodes".cm.axisCommand.cathodeAlignTableAxisY1.posAbsolute[2] := #_w1;
END_REGION

REGION Network 186: CmCathodeAlignTableAxisY1 Position Absolute Position3
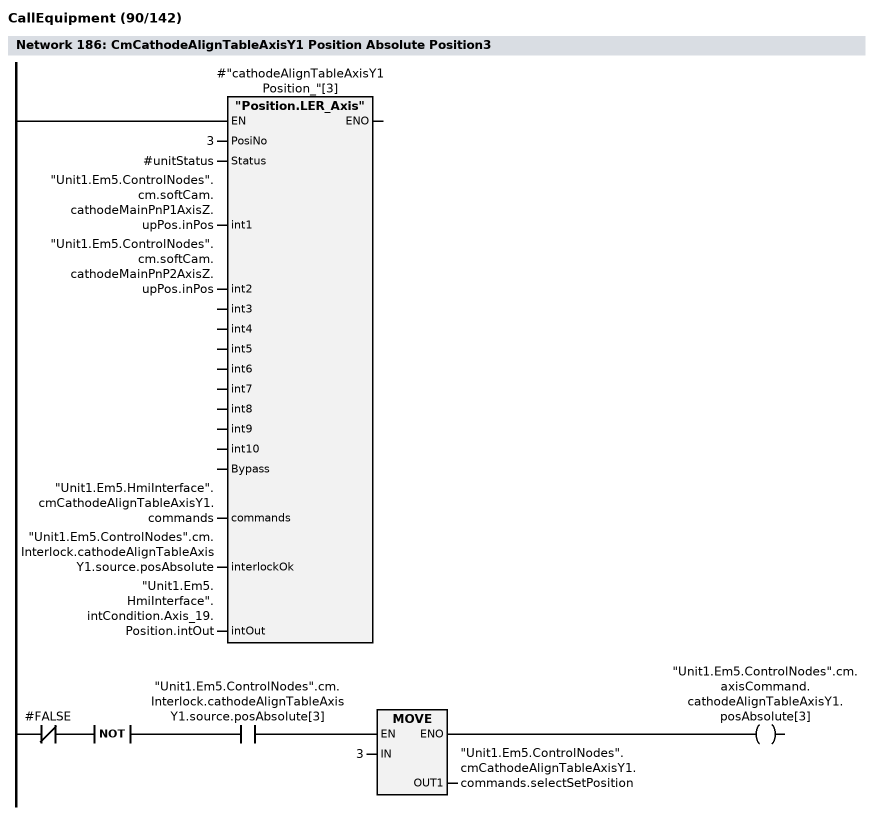
   RUNG wire#powerrail
      #"cathodeAlignTableAxisY1 Position_"[3](PosiNo := 3, Status := #unitStatus, int1 := "Unit1.Em5.ControlNodes".cm.softCam.cathodeMainPnP1AxisZ.upPos.inPos, int2 := "Unit1.Em5.ControlNodes".cm.softCam.cathodeMainPnP2AxisZ.upPos.inPos, int3 :=, int4 :=, int5 :=, int6 :=, int7 :=, int8 :=, int9 :=, int10 :=, Bypass :=, commands := "Unit1.Em5.HmiInterface".cmCathodeAlignTableAxisY1.commands, interlockOk := "Unit1.Em5.ControlNodes".cm.Interlock.cathodeAlignTableAxisY1.source.posAbsolute, intOut := "Unit1.Em5.HmiInterface".intCondition.Axis_19.Position.intOut)
   END_RUNG
   RUNG wire#powerrail
      I_Contact( #FALSE )
      Not()
      Contact( "Unit1.Em5.ControlNodes".cm.Interlock.cathodeAlignTableAxisY1.source.posAbsolute[3] )
      Move(in := 3, out1 => "Unit1.Em5.ControlNodes".cmCathodeAlignTableAxisY1.commands.selectSetPosition)
      Coil( "Unit1.Em5.ControlNodes".cm.axisCommand.cathodeAlignTableAxisY1.posAbsolute[3] )
   END_RUNG
   // the same network as SCL:
   #"cathodeAlignTableAxisY1 Position_"[3](PosiNo := 3,   // "Position.LER_Axis"
                           Status := #unitStatus,
                           int1 := "Unit1.Em5.ControlNodes".cm.softCam.cathodeMainPnP1AxisZ.upPos.inPos,
                           int2 := "Unit1.Em5.ControlNodes".cm.softCam.cathodeMainPnP2AxisZ.upPos.inPos,
                           commands := "Unit1.Em5.HmiInterface".cmCathodeAlignTableAxisY1.commands,
                           interlockOk := "Unit1.Em5.ControlNodes".cm.Interlock.cathodeAlignTableAxisY1.source.posAbsolute,
                           intOut := "Unit1.Em5.HmiInterface".intCondition.Axis_19.Position.intOut);
   #_w1 := NOT (NOT #FALSE) AND "Unit1.Em5.ControlNodes".cm.Interlock.cathodeAlignTableAxisY1.source.posAbsolute[3];
   IF #_w1 THEN "Unit1.Em5.ControlNodes".cmCathodeAlignTableAxisY1.commands.selectSetPosition := 3; END_IF;
   "Unit1.Em5.ControlNodes".cm.axisCommand.cathodeAlignTableAxisY1.posAbsolute[3] := #_w1;
END_REGION

REGION Network 187: CmCathodeAlignTableAxisY1 Position Absolute Position4
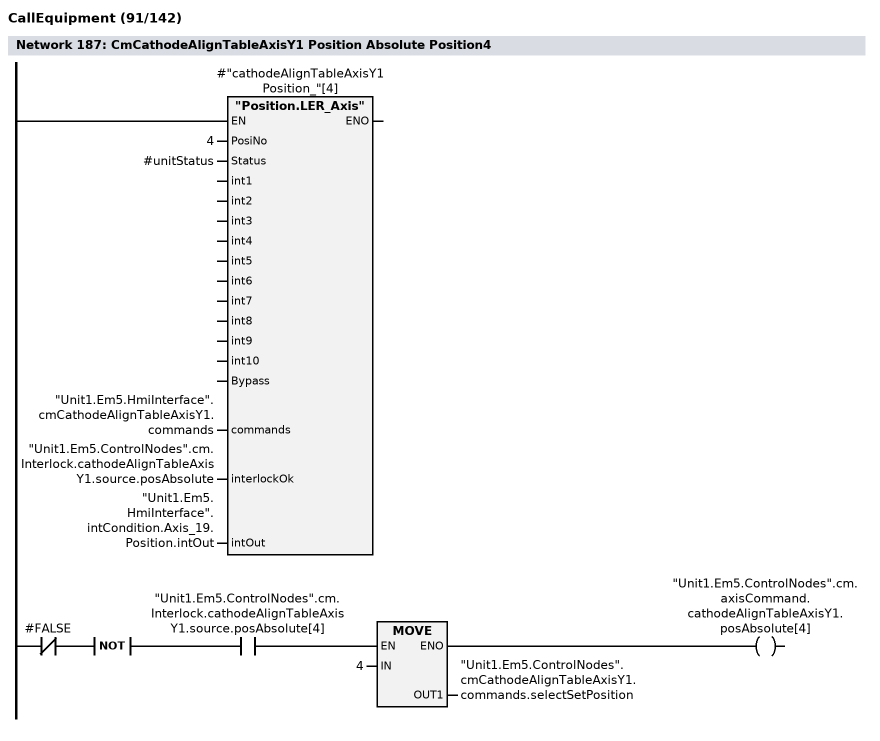
   RUNG wire#powerrail
      #"cathodeAlignTableAxisY1 Position_"[4](PosiNo := 4, Status := #unitStatus, int1 :=, int2 :=, int3 :=, int4 :=, int5 :=, int6 :=, int7 :=, int8 :=, int9 :=, int10 :=, Bypass :=, commands := "Unit1.Em5.HmiInterface".cmCathodeAlignTableAxisY1.commands, interlockOk := "Unit1.Em5.ControlNodes".cm.Interlock.cathodeAlignTableAxisY1.source.posAbsolute, intOut := "Unit1.Em5.HmiInterface".intCondition.Axis_19.Position.intOut)
   END_RUNG
   RUNG wire#powerrail
      I_Contact( #FALSE )
      Not()
      Contact( "Unit1.Em5.ControlNodes".cm.Interlock.cathodeAlignTableAxisY1.source.posAbsolute[4] )
      Move(in := 4, out1 => "Unit1.Em5.ControlNodes".cmCathodeAlignTableAxisY1.commands.selectSetPosition)
      Coil( "Unit1.Em5.ControlNodes".cm.axisCommand.cathodeAlignTableAxisY1.posAbsolute[4] )
   END_RUNG
   // the same network as SCL:
   #"cathodeAlignTableAxisY1 Position_"[4](PosiNo := 4,   // "Position.LER_Axis"
                           Status := #unitStatus,
                           commands := "Unit1.Em5.HmiInterface".cmCathodeAlignTableAxisY1.commands,
                           interlockOk := "Unit1.Em5.ControlNodes".cm.Interlock.cathodeAlignTableAxisY1.source.posAbsolute,
                           intOut := "Unit1.Em5.HmiInterface".intCondition.Axis_19.Position.intOut);
   #_w1 := NOT (NOT #FALSE) AND "Unit1.Em5.ControlNodes".cm.Interlock.cathodeAlignTableAxisY1.source.posAbsolute[4];
   IF #_w1 THEN "Unit1.Em5.ControlNodes".cmCathodeAlignTableAxisY1.commands.selectSetPosition := 4; END_IF;
   "Unit1.Em5.ControlNodes".cm.axisCommand.cathodeAlignTableAxisY1.posAbsolute[4] := #_w1;
END_REGION

REGION Network 188: CmCathodeAlignTableAxisY1 Position Absolute Position5
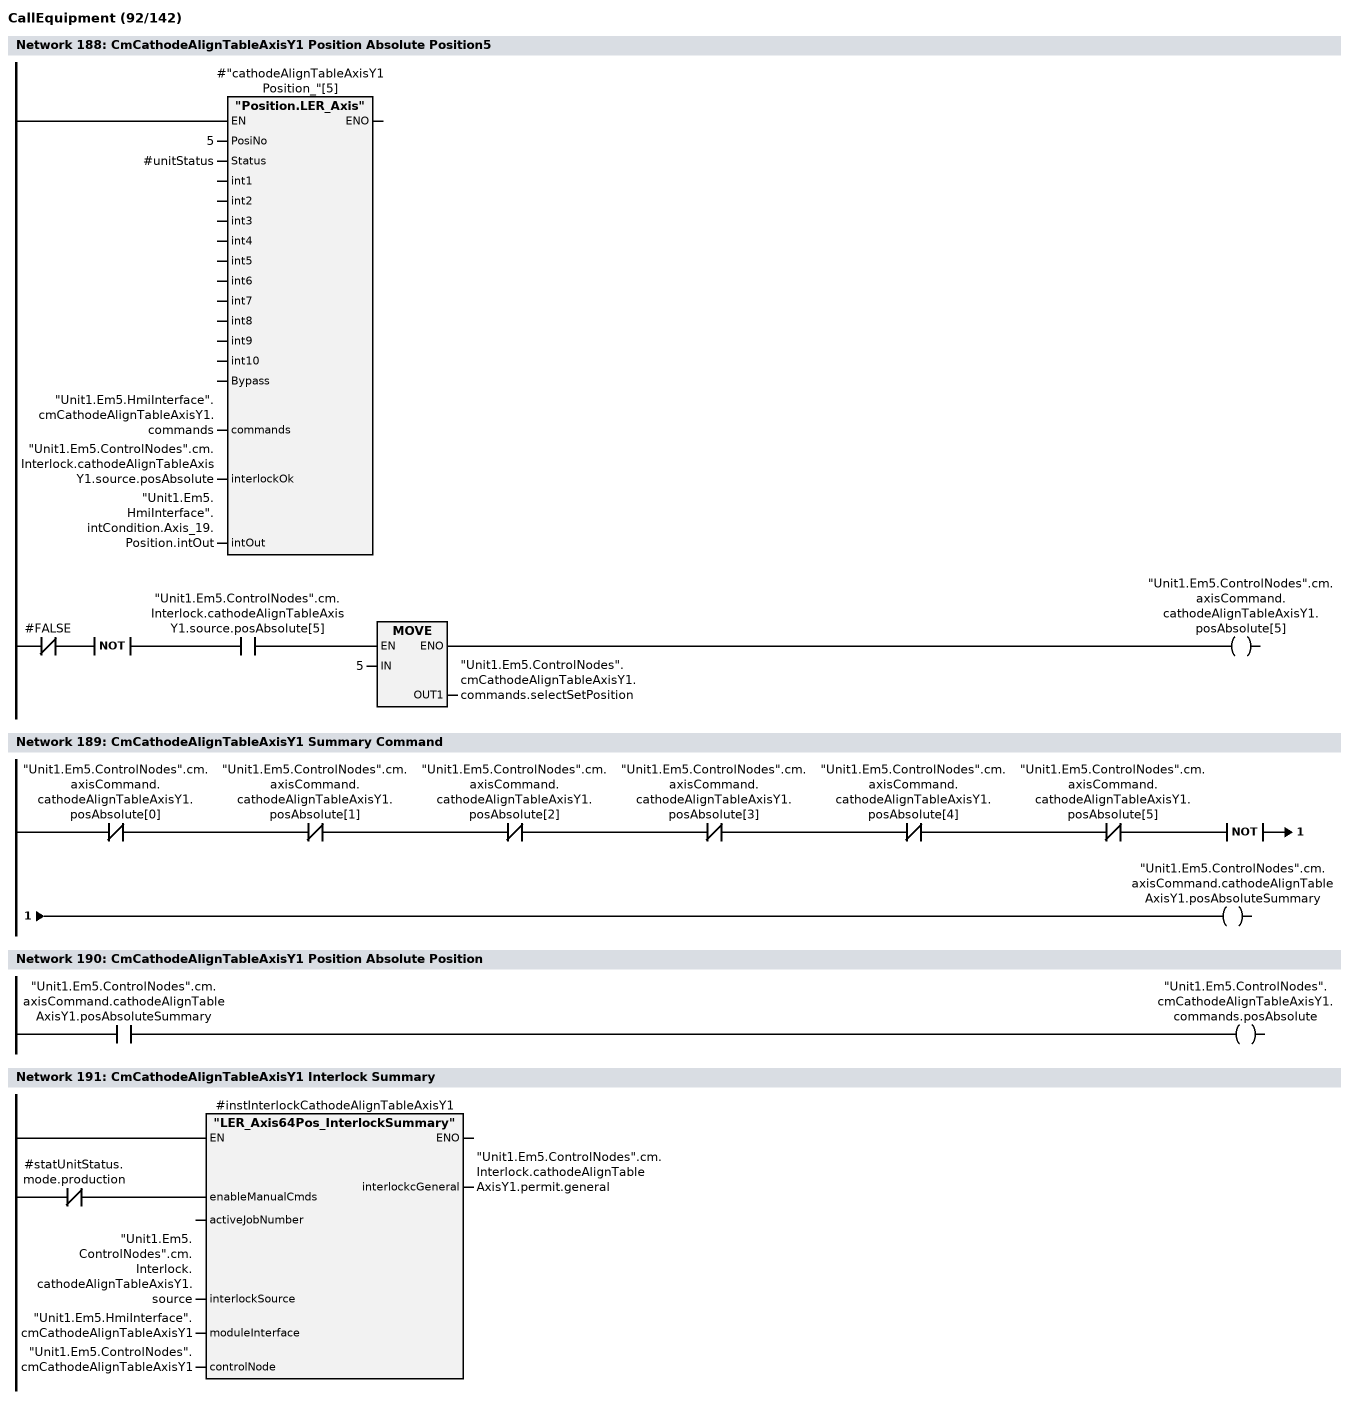
   RUNG wire#powerrail
      #"cathodeAlignTableAxisY1 Position_"[5](PosiNo := 5, Status := #unitStatus, int1 :=, int2 :=, int3 :=, int4 :=, int5 :=, int6 :=, int7 :=, int8 :=, int9 :=, int10 :=, Bypass :=, commands := "Unit1.Em5.HmiInterface".cmCathodeAlignTableAxisY1.commands, interlockOk := "Unit1.Em5.ControlNodes".cm.Interlock.cathodeAlignTableAxisY1.source.posAbsolute, intOut := "Unit1.Em5.HmiInterface".intCondition.Axis_19.Position.intOut)
   END_RUNG
   RUNG wire#powerrail
      I_Contact( #FALSE )
      Not()
      Contact( "Unit1.Em5.ControlNodes".cm.Interlock.cathodeAlignTableAxisY1.source.posAbsolute[5] )
      Move(in := 5, out1 => "Unit1.Em5.ControlNodes".cmCathodeAlignTableAxisY1.commands.selectSetPosition)
      Coil( "Unit1.Em5.ControlNodes".cm.axisCommand.cathodeAlignTableAxisY1.posAbsolute[5] )
   END_RUNG
   // the same network as SCL:
   #"cathodeAlignTableAxisY1 Position_"[5](PosiNo := 5,   // "Position.LER_Axis"
                           Status := #unitStatus,
                           commands := "Unit1.Em5.HmiInterface".cmCathodeAlignTableAxisY1.commands,
                           interlockOk := "Unit1.Em5.ControlNodes".cm.Interlock.cathodeAlignTableAxisY1.source.posAbsolute,
                           intOut := "Unit1.Em5.HmiInterface".intCondition.Axis_19.Position.intOut);
   #_w1 := NOT (NOT #FALSE) AND "Unit1.Em5.ControlNodes".cm.Interlock.cathodeAlignTableAxisY1.source.posAbsolute[5];
   IF #_w1 THEN "Unit1.Em5.ControlNodes".cmCathodeAlignTableAxisY1.commands.selectSetPosition := 5; END_IF;
   "Unit1.Em5.ControlNodes".cm.axisCommand.cathodeAlignTableAxisY1.posAbsolute[5] := #_w1;
END_REGION

REGION Network 189: CmCathodeAlignTableAxisY1 Summary Command
   RUNG wire#powerrail
      I_Contact( "Unit1.Em5.ControlNodes".cm.axisCommand.cathodeAlignTableAxisY1.posAbsolute[0] )
      I_Contact( "Unit1.Em5.ControlNodes".cm.axisCommand.cathodeAlignTableAxisY1.posAbsolute[1] )
      I_Contact( "Unit1.Em5.ControlNodes".cm.axisCommand.cathodeAlignTableAxisY1.posAbsolute[2] )
      I_Contact( "Unit1.Em5.ControlNodes".cm.axisCommand.cathodeAlignTableAxisY1.posAbsolute[3] )
      I_Contact( "Unit1.Em5.ControlNodes".cm.axisCommand.cathodeAlignTableAxisY1.posAbsolute[4] )
      I_Contact( "Unit1.Em5.ControlNodes".cm.axisCommand.cathodeAlignTableAxisY1.posAbsolute[5] )
      Not()
      Coil( "Unit1.Em5.ControlNodes".cm.axisCommand.cathodeAlignTableAxisY1.posAbsoluteSummary )
   END_RUNG
   // the same network as SCL:
   "Unit1.Em5.ControlNodes".cm.axisCommand.cathodeAlignTableAxisY1.posAbsoluteSummary := NOT (NOT "Unit1.Em5.ControlNodes".cm.axisCommand.cathodeAlignTableAxisY1.posAbsolute[0] AND NOT "Unit1.Em5.ControlNodes".cm.axisCommand.cathodeAlignTableAxisY1.posAbsolute[1] AND NOT "Unit1.Em5.ControlNodes".cm.axisCommand.cathodeAlignTableAxisY1.posAbsolute[2] AND NOT "Unit1.Em5.ControlNodes".cm.axisCommand.cathodeAlignTableAxisY1.posAbsolute[3] AND NOT "Unit1.Em5.ControlNodes".cm.axisCommand.cathodeAlignTableAxisY1.posAbsolute[4] AND NOT "Unit1.Em5.ControlNodes".cm.axisCommand.cathodeAlignTableAxisY1.posAbsolute[5]);
END_REGION

REGION Network 190: CmCathodeAlignTableAxisY1 Position Absolute Position
   RUNG wire#powerrail
      Contact( "Unit1.Em5.ControlNodes".cm.axisCommand.cathodeAlignTableAxisY1.posAbsoluteSummary )
      Coil( "Unit1.Em5.ControlNodes".cmCathodeAlignTableAxisY1.commands.posAbsolute )
   END_RUNG
   // the same network as SCL:
   "Unit1.Em5.ControlNodes".cmCathodeAlignTableAxisY1.commands.posAbsolute := "Unit1.Em5.ControlNodes".cm.axisCommand.cathodeAlignTableAxisY1.posAbsoluteSummary;
END_REGION

REGION Network 191: CmCathodeAlignTableAxisY1 Interlock Summary
   RUNG wire#powerrail
      #instInterlockCathodeAlignTableAxisY1(enableManualCmds := wire#w1, activeJobNumber :=, interlockSource := "Unit1.Em5.ControlNodes".cm.Interlock.cathodeAlignTableAxisY1.source, moduleInterface := "Unit1.Em5.HmiInterface".cmCathodeAlignTableAxisY1, controlNode := "Unit1.Em5.ControlNodes".cmCathodeAlignTableAxisY1, interlockcGeneral => "Unit1.Em5.ControlNodes".cm.Interlock.cathodeAlignTableAxisY1.permit.general)
   END_RUNG
   RUNG wire#powerrail
      I_Contact( #statUnitStatus.mode.production )
   END_RUNG wire#w1
   // the same network as SCL:
   #instInterlockCathodeAlignTableAxisY1(enableManualCmds := NOT #statUnitStatus.mode.production,   // "LER_Axis64Pos_InterlockSummary"
                           interlockSource := "Unit1.Em5.ControlNodes".cm.Interlock.cathodeAlignTableAxisY1.source,
                           moduleInterface := "Unit1.Em5.HmiInterface".cmCathodeAlignTableAxisY1,
                           controlNode := "Unit1.Em5.ControlNodes".cmCathodeAlignTableAxisY1,
                           interlockcGeneral => "Unit1.Em5.ControlNodes".cm.Interlock.cathodeAlignTableAxisY1.permit.general);
END_REGION

REGION Network 192: CmCathodeAlignTableAxisY1 velocity/speed
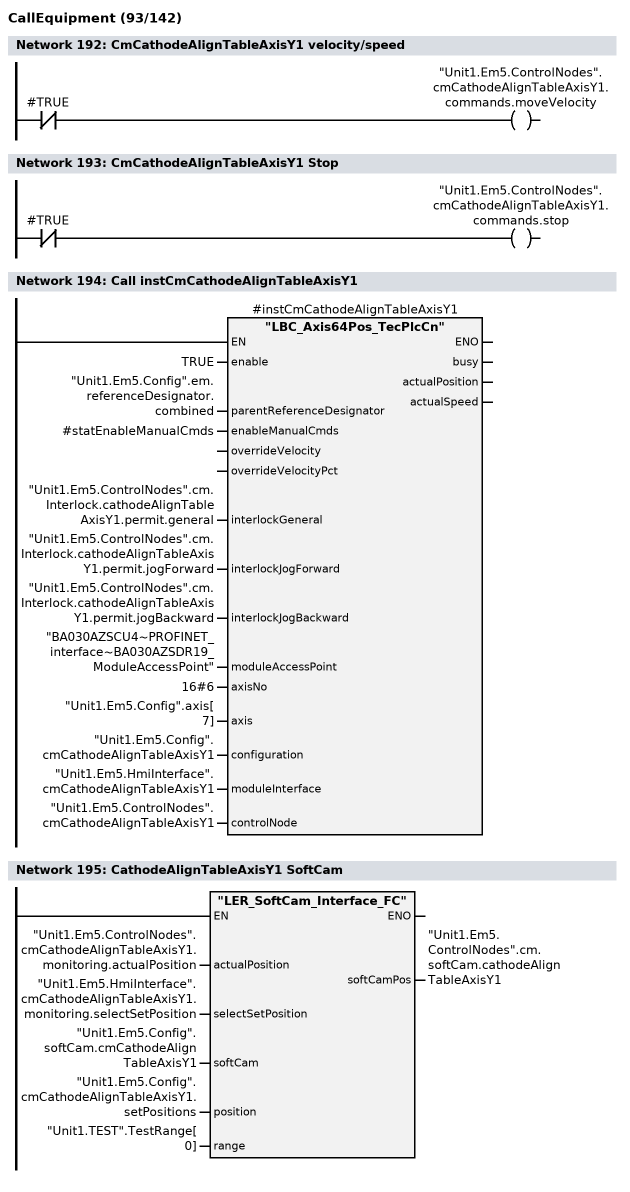
   RUNG wire#powerrail
      I_Contact( #TRUE )
      Coil( "Unit1.Em5.ControlNodes".cmCathodeAlignTableAxisY1.commands.moveVelocity )
   END_RUNG
   // the same network as SCL:
   "Unit1.Em5.ControlNodes".cmCathodeAlignTableAxisY1.commands.moveVelocity := NOT #TRUE;
END_REGION

REGION Network 193: CmCathodeAlignTableAxisY1 Stop
   RUNG wire#powerrail
      I_Contact( #TRUE )
      Coil( "Unit1.Em5.ControlNodes".cmCathodeAlignTableAxisY1.commands.stop )
   END_RUNG
   // the same network as SCL:
   "Unit1.Em5.ControlNodes".cmCathodeAlignTableAxisY1.commands.stop := NOT #TRUE;
END_REGION

REGION Network 194: Call instCmCathodeAlignTableAxisY1
   RUNG wire#powerrail
      #instCmCathodeAlignTableAxisY1(enable := TRUE, parentReferenceDesignator := "Unit1.Em5.Config".em.referenceDesignator.combined, enableManualCmds := #statEnableManualCmds, overrideVelocity :=, overrideVelocityPct :=, interlockGeneral := "Unit1.Em5.ControlNodes".cm.Interlock.cathodeAlignTableAxisY1.permit.general, interlockJogForward := "Unit1.Em5.ControlNodes".cm.Interlock.cathodeAlignTableAxisY1.permit.jogForward, interlockJogBackward := "Unit1.Em5.ControlNodes".cm.Interlock.cathodeAlignTableAxisY1.permit.jogBackward, moduleAccessPoint := "BA030AZSCU4~PROFINET_interface~BA030AZSDR19_ModuleAccessPoint", axisNo := 16#6, axis := "Unit1.Em5.Config".axis[7], configuration := "Unit1.Em5.Config".cmCathodeAlignTableAxisY1, moduleInterface := "Unit1.Em5.HmiInterface".cmCathodeAlignTableAxisY1, controlNode := "Unit1.Em5.ControlNodes".cmCathodeAlignTableAxisY1, busy =>, actualPosition =>, actualSpeed =>)
   END_RUNG
   // the same network as SCL:
   #instCmCathodeAlignTableAxisY1(enable := TRUE,   // "LBC_Axis64Pos_TecPlcCn"
                           parentReferenceDesignator := "Unit1.Em5.Config".em.referenceDesignator.combined,
                           enableManualCmds := #statEnableManualCmds,
                           interlockGeneral := "Unit1.Em5.ControlNodes".cm.Interlock.cathodeAlignTableAxisY1.permit.general,
                           interlockJogForward := "Unit1.Em5.ControlNodes".cm.Interlock.cathodeAlignTableAxisY1.permit.jogForward,
                           interlockJogBackward := "Unit1.Em5.ControlNodes".cm.Interlock.cathodeAlignTableAxisY1.permit.jogBackward,
                           moduleAccessPoint := "BA030AZSCU4~PROFINET_interface~BA030AZSDR19_ModuleAccessPoint",
                           axisNo := 16#6,
                           axis := "Unit1.Em5.Config".axis[7],
                           configuration := "Unit1.Em5.Config".cmCathodeAlignTableAxisY1,
                           moduleInterface := "Unit1.Em5.HmiInterface".cmCathodeAlignTableAxisY1,
                           controlNode := "Unit1.Em5.ControlNodes".cmCathodeAlignTableAxisY1);
END_REGION

REGION Network 195: CathodeAlignTableAxisY1 SoftCam
   RUNG wire#powerrail
      "LER_SoftCam_Interface_FC"(actualPosition := "Unit1.Em5.ControlNodes".cmCathodeAlignTableAxisY1.monitoring.actualPosition, selectSetPosition := "Unit1.Em5.HmiInterface".cmCathodeAlignTableAxisY1.monitoring.selectSetPosition, softCam := "Unit1.Em5.Config".softCam.cmCathodeAlignTableAxisY1, position := "Unit1.Em5.Config".cmCathodeAlignTableAxisY1.setPositions, range := "Unit1.TEST".TestRange[0], softCamPos => "Unit1.Em5.ControlNodes".cm.softCam.cathodeAlignTableAxisY1)
   END_RUNG
   // the same network as SCL:
   "LER_SoftCam_Interface_FC"(actualPosition := "Unit1.Em5.ControlNodes".cmCathodeAlignTableAxisY1.monitoring.actualPosition,
                           selectSetPosition := "Unit1.Em5.HmiInterface".cmCathodeAlignTableAxisY1.monitoring.selectSetPosition,
                           softCam := "Unit1.Em5.Config".softCam.cmCathodeAlignTableAxisY1,
                           position := "Unit1.Em5.Config".cmCathodeAlignTableAxisY1.setPositions,
                           range := "Unit1.TEST".TestRange[0],
                           softCamPos => "Unit1.Em5.ControlNodes".cm.softCam.cathodeAlignTableAxisY1);
END_REGION

REGION Network 197: CmAnodeAlignTableAxisY2 Enable
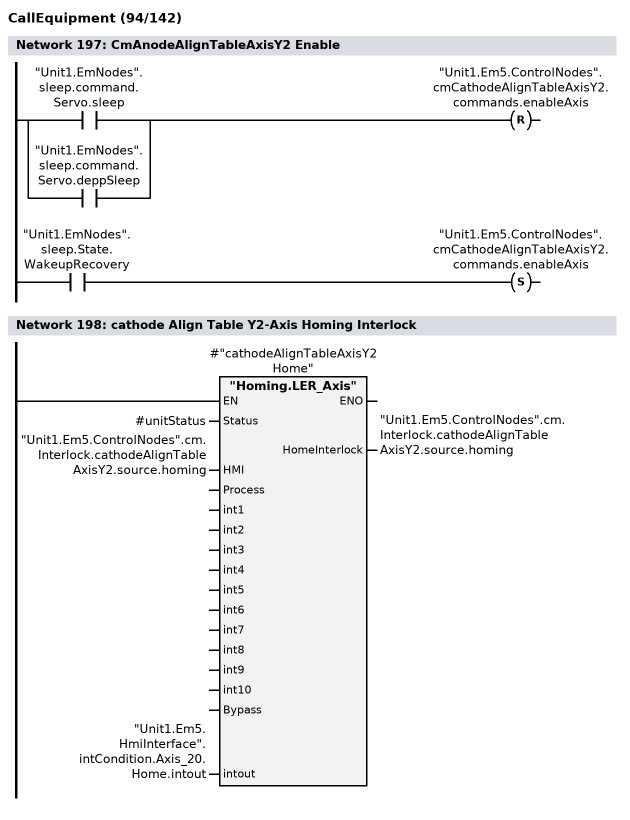
   RUNG wire#powerrail
      Contact( "Unit1.EmNodes".sleep.command.Servo.sleep )
      wire#w1
      R_Coil( "Unit1.Em5.ControlNodes".cmCathodeAlignTableAxisY2.commands.enableAxis )
   END_RUNG
   RUNG wire#powerrail
      Contact( "Unit1.EmNodes".sleep.command.Servo.deppSleep )
   END_RUNG wire#w1
   RUNG wire#powerrail
      Contact( "Unit1.EmNodes".sleep.State.WakeupRecovery )
      S_Coil( "Unit1.Em5.ControlNodes".cmCathodeAlignTableAxisY2.commands.enableAxis )
   END_RUNG
   // the same network as SCL:
   IF "Unit1.EmNodes".sleep.command.Servo.sleep OR "Unit1.EmNodes".sleep.command.Servo.deppSleep THEN
       "Unit1.Em5.ControlNodes".cmCathodeAlignTableAxisY2.commands.enableAxis := FALSE;
   END_IF;
   IF "Unit1.EmNodes".sleep.State.WakeupRecovery THEN
       "Unit1.Em5.ControlNodes".cmCathodeAlignTableAxisY2.commands.enableAxis := TRUE;
   END_IF;
END_REGION

REGION Network 198: cathode Align Table Y2-Axis Homing Interlock
   RUNG wire#powerrail
      #"cathodeAlignTableAxisY2 Home"(Status := #unitStatus, HMI := "Unit1.Em5.ControlNodes".cm.Interlock.cathodeAlignTableAxisY2.source.homing, Process :=, int1 :=, int2 :=, int3 :=, int4 :=, int5 :=, int6 :=, int7 :=, int8 :=, int9 :=, int10 :=, Bypass :=, intout := "Unit1.Em5.HmiInterface".intCondition.Axis_20.Home.intout, HomeInterlock => "Unit1.Em5.ControlNodes".cm.Interlock.cathodeAlignTableAxisY2.source.homing)
   END_RUNG
   // the same network as SCL:
   #"cathodeAlignTableAxisY2 Home"(Status := #unitStatus,   // "Homing.LER_Axis"
                           HMI := "Unit1.Em5.ControlNodes".cm.Interlock.cathodeAlignTableAxisY2.source.homing,
                           intout := "Unit1.Em5.HmiInterface".intCondition.Axis_20.Home.intout,
                           HomeInterlock => "Unit1.Em5.ControlNodes".cm.Interlock.cathodeAlignTableAxisY2.source.homing);
END_REGION

REGION Network 199: CmCathodeAlignTableAxisY2 Position Absolute Jog
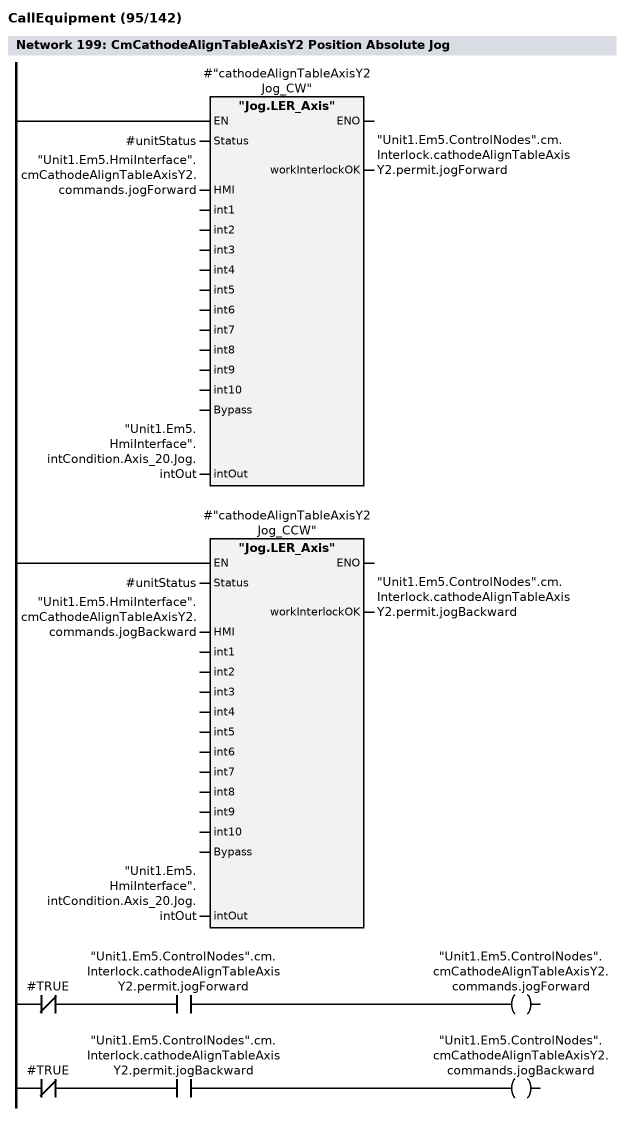
   RUNG wire#powerrail
      #"cathodeAlignTableAxisY2 Jog_CW"(Status := #unitStatus, HMI := "Unit1.Em5.HmiInterface".cmCathodeAlignTableAxisY2.commands.jogForward, int1 :=, int2 :=, int3 :=, int4 :=, int5 :=, int6 :=, int7 :=, int8 :=, int9 :=, int10 :=, Bypass :=, intOut := "Unit1.Em5.HmiInterface".intCondition.Axis_20.Jog.intOut, workInterlockOK => "Unit1.Em5.ControlNodes".cm.Interlock.cathodeAlignTableAxisY2.permit.jogForward)
   END_RUNG
   RUNG wire#powerrail
      #"cathodeAlignTableAxisY2 Jog_CCW"(Status := #unitStatus, HMI := "Unit1.Em5.HmiInterface".cmCathodeAlignTableAxisY2.commands.jogBackward, int1 :=, int2 :=, int3 :=, int4 :=, int5 :=, int6 :=, int7 :=, int8 :=, int9 :=, int10 :=, Bypass :=, intOut := "Unit1.Em5.HmiInterface".intCondition.Axis_20.Jog.intOut, workInterlockOK => "Unit1.Em5.ControlNodes".cm.Interlock.cathodeAlignTableAxisY2.permit.jogBackward)
   END_RUNG
   RUNG wire#powerrail
      I_Contact( #TRUE )
      Contact( "Unit1.Em5.ControlNodes".cm.Interlock.cathodeAlignTableAxisY2.permit.jogForward )
      Coil( "Unit1.Em5.ControlNodes".cmCathodeAlignTableAxisY2.commands.jogForward )
   END_RUNG
   RUNG wire#powerrail
      I_Contact( #TRUE )
      Contact( "Unit1.Em5.ControlNodes".cm.Interlock.cathodeAlignTableAxisY2.permit.jogBackward )
      Coil( "Unit1.Em5.ControlNodes".cmCathodeAlignTableAxisY2.commands.jogBackward )
   END_RUNG
   // the same network as SCL:
   #"cathodeAlignTableAxisY2 Jog_CW"(Status := #unitStatus,   // "Jog.LER_Axis"
                           HMI := "Unit1.Em5.HmiInterface".cmCathodeAlignTableAxisY2.commands.jogForward,
                           intOut := "Unit1.Em5.HmiInterface".intCondition.Axis_20.Jog.intOut,
                           workInterlockOK => "Unit1.Em5.ControlNodes".cm.Interlock.cathodeAlignTableAxisY2.permit.jogForward);
   #"cathodeAlignTableAxisY2 Jog_CCW"(Status := #unitStatus,   // "Jog.LER_Axis"
                           HMI := "Unit1.Em5.HmiInterface".cmCathodeAlignTableAxisY2.commands.jogBackward,
                           intOut := "Unit1.Em5.HmiInterface".intCondition.Axis_20.Jog.intOut,
                           workInterlockOK => "Unit1.Em5.ControlNodes".cm.Interlock.cathodeAlignTableAxisY2.permit.jogBackward);
   "Unit1.Em5.ControlNodes".cmCathodeAlignTableAxisY2.commands.jogForward := NOT #TRUE AND "Unit1.Em5.ControlNodes".cm.Interlock.cathodeAlignTableAxisY2.permit.jogForward;
   "Unit1.Em5.ControlNodes".cmCathodeAlignTableAxisY2.commands.jogBackward := NOT #TRUE AND "Unit1.Em5.ControlNodes".cm.Interlock.cathodeAlignTableAxisY2.permit.jogBackward;
END_REGION

REGION Network 200: CmCathodeAlignTableAxisY2 Position Absolute Position0
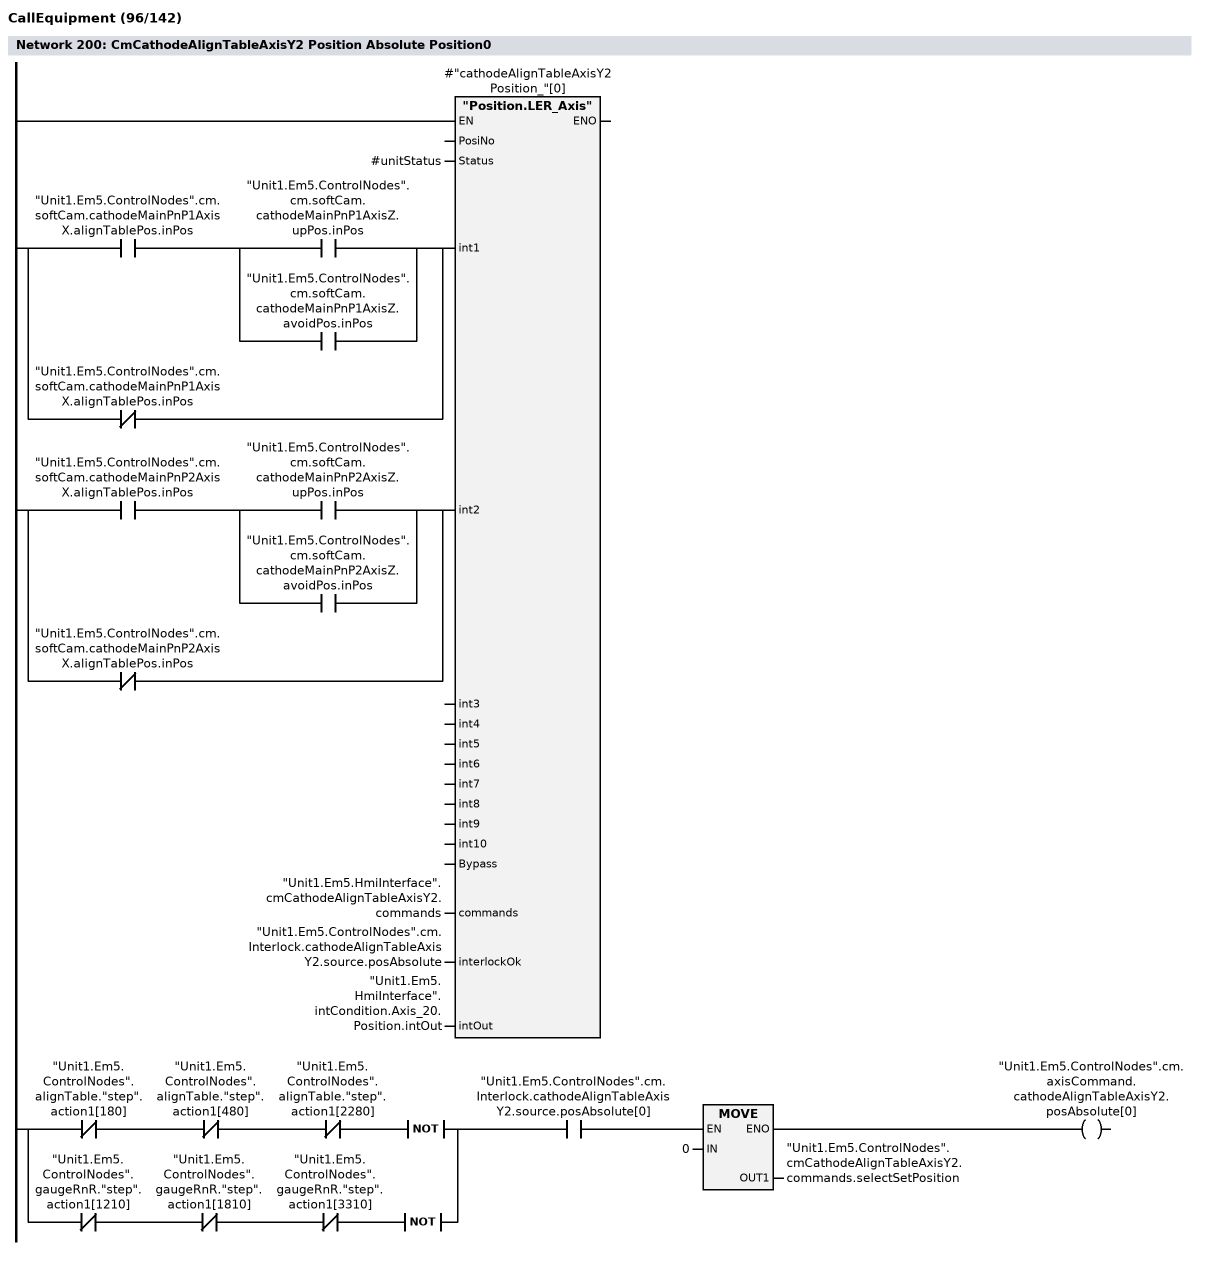
   RUNG wire#powerrail
      #"cathodeAlignTableAxisY2 Position_"[0](int1 := wire#w2, int2 := wire#w4, PosiNo :=, Status := #unitStatus, int3 :=, int4 :=, int5 :=, int6 :=, int7 :=, int8 :=, int9 :=, int10 :=, Bypass :=, commands := "Unit1.Em5.HmiInterface".cmCathodeAlignTableAxisY2.commands, interlockOk := "Unit1.Em5.ControlNodes".cm.Interlock.cathodeAlignTableAxisY2.source.posAbsolute, intOut := "Unit1.Em5.HmiInterface".intCondition.Axis_20.Position.intOut)
   END_RUNG
   RUNG wire#powerrail
      Contact( "Unit1.Em5.ControlNodes".cm.softCam.cathodeMainPnP1AxisX.alignTablePos.inPos )
      wire#w1
      Contact( "Unit1.Em5.ControlNodes".cm.softCam.cathodeMainPnP1AxisZ.upPos.inPos )
   END_RUNG wire#w2
   RUNG wire#w1
      Contact( "Unit1.Em5.ControlNodes".cm.softCam.cathodeMainPnP1AxisZ.avoidPos.inPos )
   END_RUNG wire#w2
   RUNG wire#powerrail
      I_Contact( "Unit1.Em5.ControlNodes".cm.softCam.cathodeMainPnP1AxisX.alignTablePos.inPos )
   END_RUNG wire#w2
   RUNG wire#powerrail
      Contact( "Unit1.Em5.ControlNodes".cm.softCam.cathodeMainPnP2AxisX.alignTablePos.inPos )
      wire#w3
      Contact( "Unit1.Em5.ControlNodes".cm.softCam.cathodeMainPnP2AxisZ.upPos.inPos )
   END_RUNG wire#w4
   RUNG wire#w3
      Contact( "Unit1.Em5.ControlNodes".cm.softCam.cathodeMainPnP2AxisZ.avoidPos.inPos )
   END_RUNG wire#w4
   RUNG wire#powerrail
      I_Contact( "Unit1.Em5.ControlNodes".cm.softCam.cathodeMainPnP2AxisX.alignTablePos.inPos )
   END_RUNG wire#w4
   RUNG wire#powerrail
      I_Contact( "Unit1.Em5.ControlNodes".alignTable."step".action1[180] )
      I_Contact( "Unit1.Em5.ControlNodes".alignTable."step".action1[480] )
      I_Contact( "Unit1.Em5.ControlNodes".alignTable."step".action1[2280] )
      Not()
      wire#w5
      Contact( "Unit1.Em5.ControlNodes".cm.Interlock.cathodeAlignTableAxisY2.source.posAbsolute[0] )
      Move(in := 0, out1 => "Unit1.Em5.ControlNodes".cmCathodeAlignTableAxisY2.commands.selectSetPosition)
      Coil( "Unit1.Em5.ControlNodes".cm.axisCommand.cathodeAlignTableAxisY2.posAbsolute[0] )
   END_RUNG
   RUNG wire#powerrail
      I_Contact( "Unit1.Em5.ControlNodes".gaugeRnR."step".action1[1210] )
      I_Contact( "Unit1.Em5.ControlNodes".gaugeRnR."step".action1[1810] )
      I_Contact( "Unit1.Em5.ControlNodes".gaugeRnR."step".action1[3310] )
      Not()
   END_RUNG wire#w5
   // the same network as SCL:
   #"cathodeAlignTableAxisY2 Position_"[0](Status := #unitStatus,   // "Position.LER_Axis"
                           int1 := ("Unit1.Em5.ControlNodes".cm.softCam.cathodeMainPnP1AxisX.alignTablePos.inPos AND ("Unit1.Em5.ControlNodes".cm.softCam.cathodeMainPnP1AxisZ.upPos.inPos OR "Unit1.Em5.ControlNodes".cm.softCam.cathodeMainPnP1AxisZ.avoidPos.inPos)) OR NOT "Unit1.Em5.ControlNodes".cm.softCam.cathodeMainPnP1AxisX.alignTablePos.inPos,
                           int2 := ("Unit1.Em5.ControlNodes".cm.softCam.cathodeMainPnP2AxisX.alignTablePos.inPos AND ("Unit1.Em5.ControlNodes".cm.softCam.cathodeMainPnP2AxisZ.upPos.inPos OR "Unit1.Em5.ControlNodes".cm.softCam.cathodeMainPnP2AxisZ.avoidPos.inPos)) OR NOT "Unit1.Em5.ControlNodes".cm.softCam.cathodeMainPnP2AxisX.alignTablePos.inPos,
                           commands := "Unit1.Em5.HmiInterface".cmCathodeAlignTableAxisY2.commands,
                           interlockOk := "Unit1.Em5.ControlNodes".cm.Interlock.cathodeAlignTableAxisY2.source.posAbsolute,
                           intOut := "Unit1.Em5.HmiInterface".intCondition.Axis_20.Position.intOut);
   #_w1 := (NOT (NOT "Unit1.Em5.ControlNodes".alignTable."step".action1[180] AND NOT "Unit1.Em5.ControlNodes".alignTable."step".action1[480] AND NOT "Unit1.Em5.ControlNodes".alignTable."step".action1[2280]) OR NOT (NOT "Unit1.Em5.ControlNodes".gaugeRnR."step".action1[1210] AND NOT "Unit1.Em5.ControlNodes".gaugeRnR."step".action1[1810] AND NOT "Unit1.Em5.ControlNodes".gaugeRnR."step".action1[3310])) AND "Unit1.Em5.ControlNodes".cm.Interlock.cathodeAlignTableAxisY2.source.posAbsolute[0];
   IF #_w1 THEN "Unit1.Em5.ControlNodes".cmCathodeAlignTableAxisY2.commands.selectSetPosition := 0; END_IF;
   "Unit1.Em5.ControlNodes".cm.axisCommand.cathodeAlignTableAxisY2.posAbsolute[0] := #_w1;
END_REGION

REGION Network 201: CmCathodeAlignTableAxisY2 Position Absolute Position1
